Staubli VAL3: HM.pjx

--- HM.pjx ---
Parameters version=s7.8.2 stackSize=5000 millimeterUnit=true
Program file=JTPdemo.pgx
Program file=loadmaster0.pgx
Program file=loadmaster1.pgx
Program file=loadmaster2.pgx
Program file=loadmaster3.pgx
Program file=loadmaster4.pgx
Program file=loadmaster5.pgx
Program file=loadmaster6.pgx
Program file=loadmaster7.pgx
Program file=loadmaster8.pgx
Program file=loadmaster9.pgx
Program file=madol.pgx
Program file=oldmaduofrme.pgx
Program file=proDEMO.pgx
Program file=saveOldframe.pgx
Program file=SAVEtoolAfranme.pgx
Program file=SMOVE.pgx
Program file=start.pgx
Program file=stop.pgx
Program file=takestop.pgx
Program file=tooolAndFrame.pgx
Data file=HM.dtx
Library alias=master path=Disk://master/master.pjx
Library alias=lib path=Disk://frmtool/frmtool.pjx

--- HM.dtx ---
bool b0
bool b1 = true
bool b2
bool b3
bool b4
bool bA[10] = true
bool bPause
bool bruning
bool bstop
public dio diganying = {link=BasicIO-1\%I2}
dio distart = {link=usrIn0}
dio distop = {link=usrIn1}
dio ditab = {link=BasicIO-1\%I1}
dio dixi = {link=BasicIO-1\%I0}
dio dochui = {link=BasicIO-1\%Q0}
dio doxi = {link=BasicIO-1\%Q1}
public frame f1 = {x=112.060509, y=-257.129174, z=-98.62342, rx=-0.279882, ry=0.007961, rz=179.830294, fatherId=world[0]}
public frame frmaster[10]
  [0] = {x=487, y=64, z=-100.5, rx=5, rz=-92.998, fatherId=world[0]}
  [1] = {x=472, y=210, z=-97, rz=175, fatherId=world[0]}
  [2] = {x=472, y=201, z=-98, rx=0.5, rz=98, fatherId=world[0]}
  [3] = {fatherId=world[0]}
  [4] = {fatherId=world[0]}
  [5] = {fatherId=world[0]}
  [6] = {fatherId=world[0]}
  [7] = {x=487, y=64, z=-100.5, rx=5, rz=-92.998, fatherId=world[0]}
  [8] = {x=487, y=64, z=-100.5, rx=5, rz=-92.998, fatherId=world[0]}
  [9] = {x=487, y=64, z=-100.5, rx=5, rz=-92.998, fatherId=world[0]}
jointRx jA[20]
  [0] = {j1=-36.809158, j2=6.473103, j3=115.475326, j4=0.67904, j5=57.498227, j6=-129.910351}
  [1] = {j1=-46.642796, j2=10.279087, j3=109.084102, j4=6.799386, j5=57.689141, j6=-43.494821}
  [2] = {j1=-36.809158, j2=6.473103, j3=115.475326, j4=0.67904, j5=57.498227, j6=-129.910351}
  [3] = {j1=-46.642796, j2=10.279087, j3=109.084102, j4=6.799386, j5=57.689141, j6=-43.494821}
  [4] = {j1=-36.809158, j2=6.473103, j3=115.475326, j4=0.67904, j5=57.498227, j6=-129.910351}
  [5] = {j1=-46.642796, j2=10.279087, j3=109.084102, j4=6.799386, j5=57.689141, j6=-43.494821}
  [6] = {j1=-36.809158, j2=6.473103, j3=115.475326, j4=0.67904, j5=57.498227, j6=-129.910351}
  [7] = {j1=-46.642796, j2=10.279087, j3=109.084102, j4=6.799386, j5=57.689141, j6=-43.494821}
  [8] = {j1=-36.809158, j2=6.473103, j3=115.475326, j4=0.67904, j5=57.498227, j6=-129.910351}
  [9] = {j1=-46.642796, j2=10.279087, j3=109.084102, j4=6.799386, j5=57.689141, j6=-43.494821}
  [10] = {j1=-36.809158, j2=6.473103, j3=115.475326, j4=0.67904, j5=57.498227, j6=-129.910351}
  [11] = {j1=-46.642796, j2=10.279087, j3=109.084102, j4=6.799386, j5=57.689141, j6=-43.494821}
  [12] = {j1=-36.809158, j2=6.473103, j3=115.475326, j4=0.67904, j5=57.498227, j6=-129.910351}
  [13] = {j1=-46.642796, j2=10.279087, j3=109.084102, j4=6.799386, j5=57.689141, j6=-43.494821}
  [14] = {j1=-36.809158, j2=6.473103, j3=115.475326, j4=0.67904, j5=57.498227, j6=-129.910351}
  [15] = {j1=-46.642796, j2=10.279087, j3=109.084102, j4=6.799386, j5=57.689141, j6=-43.494821}
  [16] = {j1=-36.809158, j2=6.473103, j3=115.475326, j4=0.67904, j5=57.498227, j6=-129.910351}
  [17] = {j1=-46.642796, j2=10.279087, j3=109.084102, j4=6.799386, j5=57.689141, j6=-43.494821}
  [18] = {j1=-36.809158, j2=6.473103, j3=115.475326, j4=0.67904, j5=57.498227, j6=-129.910351}
  [19] = {j1=-46.642796, j2=10.279087, j3=109.084102, j4=6.799386, j5=57.689141, j6=-43.494821}
jointRx jXieLiao = {j1=-96.476357, j2=75.42768, j3=32.803482, j4=-0.025549, j5=71.586432, j6=-93.064419}
jointRx jbegin = {j1=-36.809158, j2=6.473103, j3=115.475326, j4=0.67904, j5=57.498227, j6=-129.910351}
jointRx jchack = {j1=-102.590963, j2=19.158438, j3=101.614955, j4=-0.038681, j5=59.106199, j6=77.212336}
jointRx jend = {j1=-46.642796, j2=10.279087, j3=109.084102, j4=6.799386, j5=57.689141, j6=-43.494821}
jointRx jf = {j1=-96.478721, j2=69.604961, j3=32.597072, j4=-0.024894, j5=77.614683, j6=-93.069451}
jointRx jready = {j1=-93.60071, j2=14.149819, j3=120.13944, j4=-0.061569, j5=45.526614, j6=86.705521}
jointRx jstart = {j1=-102.590964, j2=19.158205, j3=101.615123, j4=-0.038768, j5=59.105849, j6=77.212673}
mdesc m1
mdesc mFast
mdesc mSuDu[3]
  [0] = {leave=0.5, reach=0.5}
  [1] = {leave=0.5, reach=0.5}
  [2] = {leave=0.5, reach=0.5}
num n0 = 1
num n1 = 2
num n2
num nJTP
num nPY = 320
num nPYB
num nPYC = 320
num nPYtest = -0.957
num nPeak0[3]
  [0] = 66
  [1] = 198
num nPeak1[4]
  [0] = 193
  [1] = 359
  [2] = 551
num nPeak2
num nPeak3
num nPeak4
num nPeak5
num nPeak6
num nPeak7
num nPeak8
num nPeak9
num nc
num ndemo = 263
num nframe = 10
num nframeSave[10]
  [1] = 1
  [2] = 2
  [3] = 3
  [4] = 4
  [5] = 5
  [6] = 6
num ni
num ninttool = 10
num nmaster = 263
num nsize[10]
  [0] = 263
  [1] = 713
  [2] = 1183
num ntool = 10
num ntoolSave[10]
  [1] = 1
  [2] = 2
  [3] = 3
  [4] = 4
pointRx p1 = {x=0.01979, y=0.014228, z=76.837612, rx=0.284492, ry=-179.996615, rz=2.95459, fatherId=f1[0]}
pointRx p2 = {x=0.019785, y=0.014249, z=0.8, rx=0.28, ry=-179.997276, rz=2.954581, fatherId=f1[0]}
pointRx pXieLiao[2]
  [0] = {x=530.900904, y=-168.692362, z=119.392812, rx=179.999348, ry=-0.000559, rz=86.125781, fatherId=f1[0]}
  [1] = {x=530.900895, y=-168.692364, z=88.853022, rx=179.999359, ry=-0.000487, rz=86.125781, fatherId=f1[0]}
pointRx pdemo0[263]
  [0] = {x=-68.939309, y=2.594876, z=125.851419, rx=-179.999842, ry=-4.539241, rz=-20.572084, shoulder=lefty, elbow=epositive, wrist=wpositive, fatherId=frmaster[0]}
  [1] = {x=-70.093865, y=2.593252, z=111.351632, rx=179.999825, ry=-4.539343, rz=-20.573264, shoulder=lefty, elbow=epositive, wrist=wpositive, fatherId=frmaster[0]}
  [2] = {x=-70.092383, y=2.592813, z=101.346658, rx=179.998902, ry=-4.539362, rz=-20.572687, shoulder=lefty, elbow=epositive, wrist=wpositive, fatherId=frmaster[0]}
  [3] = {x=-65.564746, y=4.520144, z=104.636521, rx=-179.999623, ry=-7.320234, rz=-18.950696, shoulder=lefty, elbow=epositive, wrist=wpositive, fatherId=frmaster[0]}
  [4] = {x=-62.147679, y=5.718087, z=106.809457, rx=-179.999792, ry=-9.281495, rz=-17.978552, shoulder=lefty, elbow=epositive, wrist=wpositive, fatherId=frmaster[0]}
  [5] = {x=-57.8022, y=7.018139, z=109.291144, rx=179.999693, ry=-11.675298, rz=-16.93825, shoulder=lefty, elbow=epositive, wrist=wpositive, fatherId=frmaster[0]}
  [6] = {x=-55.21006, y=7.693586, z=110.648654, rx=-179.999664, ry=-13.066514, rz=-16.401657, shoulder=lefty, elbow=epositive, wrist=wpositive, fatherId=frmaster[0]}
  [7] = {x=-52.124031, y=8.434718, z=112.144392, rx=-179.999565, ry=-14.684361, rz=-15.820245, shoulder=lefty, elbow=epositive, wrist=wpositive, fatherId=frmaster[0]}
  [8] = {x=-48.559584, y=9.194588, z=113.730853, rx=179.999704, ry=-16.519257, rz=-15.226253, shoulder=lefty, elbow=epositive, wrist=wpositive, fatherId=frmaster[0]}
  [9] = {x=-44.443282, y=9.975646, z=115.393939, rx=-179.999788, ry=-18.600614, rz=-14.619836, shoulder=lefty, elbow=epositive, wrist=wpositive, fatherId=frmaster[0]}
  [10] = {x=-39.800946, y=10.739014, z=117.055469, rx=-179.999297, ry=-20.90861, rz=-14.028689, shoulder=lefty, elbow=epositive, wrist=wpositive, fatherId=frmaster[0]}
  [11] = {x=-34.573283, y=11.490434, z=118.675732, rx=-179.999727, ry=-23.468814, rz=-13.446694, shoulder=lefty, elbow=epositive, wrist=wpositive, fatherId=frmaster[0]}
  [12] = {x=-28.795169, y=12.206445, z=120.17003, rx=-179.99997, ry=-26.259293, rz=-12.893915, shoulder=lefty, elbow=epositive, wrist=wpositive, fatherId=frmaster[0]}
  [13] = {x=-25.703845, y=12.55415, z=120.847864, rx=-179.999289, ry=-27.738767, rz=-12.625116, shoulder=lefty, elbow=epositive, wrist=wpositive, fatherId=frmaster[0]}
  [14] = {x=-22.481958, y=12.893896, z=121.46453, rx=-179.999584, ry=-29.273016, rz=-12.362705, shoulder=lefty, elbow=epositive, wrist=wpositive, fatherId=frmaster[0]}
  [15] = {x=-19.100752, y=13.220332, z=122.011165, rx=179.999554, ry=-30.873819, rz=-12.110668, shoulder=lefty, elbow=epositive, wrist=wpositive, fatherId=frmaster[0]}
  [16] = {x=-15.56624, y=13.542118, z=122.492282, rx=179.999906, ry=-32.542669, rz=-11.862432, shoulder=lefty, elbow=epositive, wrist=wpositive, fatherId=frmaster[0]}
  [17] = {x=-11.862171, y=13.86112, z=122.876566, rx=-179.999624, ry=-34.280739, rz=-11.617025, shoulder=lefty, elbow=epositive, wrist=wpositive, fatherId=frmaster[0]}
  [18] = {x=-7.999903, y=14.172788, z=123.156947, rx=-179.999236, ry=-36.08968, rz=-11.375401, shoulder=lefty, elbow=epositive, wrist=wpositive, fatherId=frmaster[0]}
  [19] = {x=-3.982068, y=14.472199, z=123.31508, rx=-179.999527, ry=-37.973145, rz=-11.146259, shoulder=lefty, elbow=epositive, wrist=wpositive, fatherId=frmaster[0]}
  [20] = {x=0.003718, y=14.757289, z=123.343316, rx=-179.999752, ry=-39.835809, rz=-10.926527, shoulder=lefty, elbow=epositive, wrist=wpositive, fatherId=frmaster[0]}
  [21] = {x=3.926135, y=15.026312, z=123.249243, rx=-179.999627, ry=-41.673849, rz=-10.71735, shoulder=lefty, elbow=epositive, wrist=wpositive, fatherId=frmaster[0]}
  [22] = {x=7.787882, y=15.285683, z=123.023611, rx=-179.999358, ry=-43.485441, rz=-10.516961, shoulder=lefty, elbow=epositive, wrist=wpositive, fatherId=frmaster[0]}
  [23] = {x=3.636586, y=13.055492, z=123.517209, rx=-179.999236, ry=-41.68691, rz=-12.371075, shoulder=lefty, elbow=epositive, wrist=wpositive, fatherId=frmaster[0]}
  [24] = {x=-0.115648, y=10.554981, z=123.842224, rx=-179.9989, ry=-40.072666, rz=-14.410733, shoulder=lefty, elbow=epositive, wrist=wpositive, fatherId=frmaster[0]}
  [25] = {x=-2.87591, y=7.781393, z=124.033861, rx=-179.999939, ry=-38.90966, rz=-16.64011, shoulder=lefty, elbow=epositive, wrist=wpositive, fatherId=frmaster[0]}
  [26] = {x=-5.00539, y=4.722334, z=124.137637, rx=-179.999391, ry=-38.009486, rz=-19.063272, shoulder=lefty, elbow=epositive, wrist=wpositive, fatherId=frmaster[0]}
  [27] = {x=-6.286632, y=1.407733, z=124.172868, rx=-179.999461, ry=-37.465687, rz=-21.663049, shoulder=lefty, elbow=epositive, wrist=wpositive, fatherId=frmaster[0]}
  [28] = {x=-6.757242, y=-1.994395, z=124.137734, rx=-179.999849, ry=-37.245975, rz=-24.324062, shoulder=lefty, elbow=epositive, wrist=wpositive, fatherId=frmaster[0]}
  [29] = {x=-6.623, y=-5.406644, z=124.030721, rx=-179.999523, ry=-37.25052, rz=-26.994443, shoulder=lefty, elbow=epositive, wrist=wpositive, fatherId=frmaster[0]}
  [30] = {x=-5.670017, y=-8.784356, z=123.866129, rx=179.999811, ry=-37.580919, rz=-29.6487, shoulder=lefty, elbow=epositive, wrist=wpositive, fatherId=frmaster[0]}
  [31] = {x=-4.463415, y=-12.188788, z=123.606311, rx=-179.999254, ry=-37.973613, rz=-32.334872, shoulder=lefty, elbow=epositive, wrist=wpositive, fatherId=frmaster[0]}
  [32] = {x=-2.488328, y=-15.635885, z=123.233005, rx=-179.999282, ry=-38.667419, rz=-35.069863, shoulder=lefty, elbow=epositive, wrist=wpositive, fatherId=frmaster[0]}
  [33] = {x=-0.694211, y=-19.173546, z=122.713263, rx=-179.99927, ry=-39.206278, rz=-37.895277, shoulder=lefty, elbow=epositive, wrist=wpositive, fatherId=frmaster[0]}
  [34] = {x=1.757246, y=-22.68427, z=122.039686, rx=179.999513, ry=-40.003209, rz=-40.732797, shoulder=lefty, elbow=epositive, wrist=wpositive, fatherId=frmaster[0]}
  [35] = {x=3.612463, y=-26.090704, z=121.2463, rx=-179.999323, ry=-40.461466, rz=-43.533179, shoulder=lefty, elbow=epositive, wrist=wpositive, fatherId=frmaster[0]}
  [36] = {x=6.005382, y=-29.344396, z=120.330355, rx=-179.999297, ry=-41.144506, rz=-46.26609, shoulder=lefty, elbow=epositive, wrist=wpositive, fatherId=frmaster[0]}
  [37] = {x=8.178744, y=-32.51397, z=119.292757, rx=-179.999423, ry=-41.674458, rz=-48.980771, shoulder=lefty, elbow=epositive, wrist=wpositive, fatherId=frmaster[0]}
  [38] = {x=10.802026, y=-35.564113, z=118.108689, rx=-179.999959, ry=-42.396715, rz=-51.657334, shoulder=lefty, elbow=epositive, wrist=wpositive, fatherId=frmaster[0]}
  [39] = {x=13.535281, y=-38.529801, z=116.777056, rx=179.9997, ry=-43.139921, rz=-54.32829, shoulder=lefty, elbow=epositive, wrist=wpositive, fatherId=frmaster[0]}
  [40] = {x=16.594916, y=-41.383811, z=115.276942, rx=-179.999131, ry=-44.02302, rz=-56.968323, shoulder=lefty, elbow=epositive, wrist=wpositive, fatherId=frmaster[0]}
  [41] = {x=19.918159, y=-44.039781, z=113.620021, rx=-179.999247, ry=-45.050326, rz=-59.514928, shoulder=lefty, elbow=epositive, wrist=wpositive, fatherId=frmaster[0]}
  [42] = {x=23.337445, y=-46.461139, z=111.840864, rx=179.999666, ry=-46.157544, rz=-61.921405, shoulder=lefty, elbow=epositive, wrist=wpositive, fatherId=frmaster[0]}
  [43] = {x=19.98531, y=-46.203057, z=112.638501, rx=-179.999542, ry=-44.473252, rz=-61.637393, shoulder=lefty, elbow=epositive, wrist=wpositive, fatherId=frmaster[0]}
  [44] = {x=16.475747, y=-45.923809, z=113.355993, rx=-179.999849, ry=-42.732145, rz=-61.337507, shoulder=lefty, elbow=epositive, wrist=wpositive, fatherId=frmaster[0]}
  [45] = {x=12.814869, y=-45.622369, z=113.989509, rx=179.999801, ry=-40.928708, rz=-61.018055, shoulder=lefty, elbow=epositive, wrist=wpositive, fatherId=frmaster[0]}
  [46] = {x=8.994815, y=-45.291604, z=114.523598, rx=-179.998902, ry=-39.065668, rz=-60.674105, shoulder=lefty, elbow=epositive, wrist=wpositive, fatherId=frmaster[0]}
  [47] = {x=5.221971, y=-44.883621, z=114.948885, rx=179.99941, ry=-37.262806, rz=-60.255183, shoulder=lefty, elbow=epositive, wrist=wpositive, fatherId=frmaster[0]}
  [48] = {x=1.449749, y=-44.426571, z=115.268039, rx=-179.999677, ry=-35.476818, rz=-59.799009, shoulder=lefty, elbow=epositive, wrist=wpositive, fatherId=frmaster[0]}
  [49] = {x=-2.30993, y=-43.925823, z=115.469722, rx=-179.999667, ry=-33.714009, rz=-59.302848, shoulder=lefty, elbow=epositive, wrist=wpositive, fatherId=frmaster[0]}
  [50] = {x=-6.054682, y=-43.371912, z=115.566057, rx=-179.99921, ry=-31.979643, rz=-58.765546, shoulder=lefty, elbow=epositive, wrist=wpositive, fatherId=frmaster[0]}
  [51] = {x=-9.706723, y=-42.74106, z=115.566586, rx=-179.999762, ry=-30.311063, rz=-58.161529, shoulder=lefty, elbow=epositive, wrist=wpositive, fatherId=frmaster[0]}
  [52] = {x=-13.324451, y=-42.074603, z=115.473731, rx=179.999869, ry=-28.675999, rz=-57.526544, shoulder=lefty, elbow=epositive, wrist=wpositive, fatherId=frmaster[0]}
  [53] = {x=-16.85983, y=-41.366634, z=115.277163, rx=179.999422, ry=-27.08369, rz=-56.861863, shoulder=lefty, elbow=epositive, wrist=wpositive, fatherId=frmaster[0]}
  [54] = {x=-20.301815, y=-40.617438, z=115.002996, rx=-179.999332, ry=-25.546739, rz=-56.16562, shoulder=lefty, elbow=epositive, wrist=wpositive, fatherId=frmaster[0]}
  [55] = {x=-26.791225, y=-38.992184, z=114.248958, rx=-179.998983, ry=-22.681622, rz=-54.674543, shoulder=lefty, elbow=epositive, wrist=wpositive, fatherId=frmaster[0]}
  [56] = {x=-32.776952, y=-37.211639, z=113.279864, rx=179.999314, ry=-20.079214, rz=-53.068219, shoulder=lefty, elbow=epositive, wrist=wpositive, fatherId=frmaster[0]}
  [57] = {x=-38.202715, y=-35.254548, z=112.201778, rx=-179.999362, ry=-17.75731, rz=-51.337224, shoulder=lefty, elbow=epositive, wrist=wpositive, fatherId=frmaster[0]}
  [58] = {x=-43.075297, y=-33.139465, z=111.069332, rx=-179.99912, ry=-15.713738, rz=-49.495669, shoulder=lefty, elbow=epositive, wrist=wpositive, fatherId=frmaster[0]}
  [59] = {x=-47.485041, y=-30.827965, z=109.907709, rx=-179.999984, ry=-13.891332, rz=-47.517107, shoulder=lefty, elbow=epositive, wrist=wpositive, fatherId=frmaster[0]}
  [60] = {x=-51.464947, y=-28.297069, z=108.771217, rx=-179.999297, ry=-12.28541, rz=-45.387575, shoulder=lefty, elbow=epositive, wrist=wpositive, fatherId=frmaster[0]}
  [61] = {x=-58.258069, y=-22.435578, z=106.618321, rx=179.999827, ry=-9.619917, rz=-40.577437, shoulder=lefty, elbow=epositive, wrist=wpositive, fatherId=frmaster[0]}
  [62] = {x=-63.471689, y=-15.637158, z=104.757087, rx=179.999576, ry=-7.611857, rz=-35.15207, shoulder=lefty, elbow=epositive, wrist=wpositive, fatherId=frmaster[0]}
  [63] = {x=-69.230412, y=-4.124169, z=101.957036, rx=-179.999606, ry=-5.040121, rz=-25.997789, shoulder=lefty, elbow=epositive, wrist=wpositive, fatherId=frmaster[0]}
  [64] = {x=-69.233338, y=-4.126295, z=111.947543, rx=179.999548, ry=-5.039948, rz=-25.997986, shoulder=lefty, elbow=epositive, wrist=wpositive, fatherId=frmaster[0]}
  [65] = {x=-67.950588, y=-4.124727, z=126.453883, rx=179.999566, ry=-5.039306, rz=-25.997643, shoulder=lefty, elbow=epositive, wrist=wpositive, fatherId=frmaster[0]}
  [66] = {x=-68.939309, y=2.594876, z=125.851419, rx=0.000158, ry=-175.460759, rz=-20.572084, shoulder=lefty, elbow=epositive, wrist=wpositive, fatherId=frmaster[0]}
  [67] = {x=-70.093865, y=2.593252, z=111.351632, rx=-0.000175, ry=-175.460657, rz=-20.573264, shoulder=lefty, elbow=epositive, wrist=wpositive, fatherId=frmaster[0]}
  [68] = {x=-70.092383, y=2.592813, z=101.346658, rx=-0.001098, ry=-175.460638, rz=-20.572687, shoulder=lefty, elbow=epositive, wrist=wpositive, fatherId=frmaster[0]}
  [69] = {x=-65.564746, y=4.520144, z=104.636521, rx=0.000377, ry=-172.679766, rz=-18.950696, shoulder=lefty, elbow=epositive, wrist=wpositive, fatherId=frmaster[0]}
  [70] = {x=-62.147679, y=5.718087, z=106.809457, rx=0.000208, ry=-170.718505, rz=-17.978552, shoulder=lefty, elbow=epositive, wrist=wpositive, fatherId=frmaster[0]}
  [71] = {x=-57.8022, y=7.018139, z=109.291144, rx=-0.000307, ry=-168.324702, rz=-16.93825, shoulder=lefty, elbow=epositive, wrist=wpositive, fatherId=frmaster[0]}
  [72] = {x=-55.21006, y=7.693586, z=110.648654, rx=0.000336, ry=-166.933486, rz=-16.401657, shoulder=lefty, elbow=epositive, wrist=wpositive, fatherId=frmaster[0]}
  [73] = {x=-52.124031, y=8.434718, z=112.144392, rx=0.000435, ry=-165.315639, rz=-15.820245, shoulder=lefty, elbow=epositive, wrist=wpositive, fatherId=frmaster[0]}
  [74] = {x=-48.559584, y=9.194588, z=113.730853, rx=-0.000296, ry=-163.480743, rz=-15.226253, shoulder=lefty, elbow=epositive, wrist=wpositive, fatherId=frmaster[0]}
  [75] = {x=-44.443282, y=9.975646, z=115.393939, rx=0.000212, ry=-161.399386, rz=-14.619836, shoulder=lefty, elbow=epositive, wrist=wpositive, fatherId=frmaster[0]}
  [76] = {x=-39.800946, y=10.739014, z=117.055469, rx=0.000703, ry=-159.09139, rz=-14.028689, shoulder=lefty, elbow=epositive, wrist=wpositive, fatherId=frmaster[0]}
  [77] = {x=-34.573283, y=11.490434, z=118.675732, rx=0.000273, ry=-156.531186, rz=-13.446694, shoulder=lefty, elbow=epositive, wrist=wpositive, fatherId=frmaster[0]}
  [78] = {x=-28.795169, y=12.206445, z=120.17003, rx=0.00003, ry=-153.740707, rz=-12.893915, shoulder=lefty, elbow=epositive, wrist=wpositive, fatherId=frmaster[0]}
  [79] = {x=-25.703845, y=12.55415, z=120.847864, rx=0.000711, ry=-152.261233, rz=-12.625116, shoulder=lefty, elbow=epositive, wrist=wpositive, fatherId=frmaster[0]}
  [80] = {x=-22.481958, y=12.893896, z=121.46453, rx=0.000416, ry=-150.726984, rz=-12.362705, shoulder=lefty, elbow=epositive, wrist=wpositive, fatherId=frmaster[0]}
  [81] = {x=-19.100752, y=13.220332, z=122.011165, rx=-0.000446, ry=-149.126181, rz=-12.110668, shoulder=lefty, elbow=epositive, wrist=wpositive, fatherId=frmaster[0]}
  [82] = {x=-15.56624, y=13.542118, z=122.492282, rx=-0.000094, ry=-147.457331, rz=-11.862432, shoulder=lefty, elbow=epositive, wrist=wpositive, fatherId=frmaster[0]}
  [83] = {x=-11.862171, y=13.86112, z=122.876566, rx=0.000376, ry=-145.719261, rz=-11.617025, shoulder=lefty, elbow=epositive, wrist=wpositive, fatherId=frmaster[0]}
  [84] = {x=-7.999903, y=14.172788, z=123.156947, rx=0.000764, ry=-143.91032, rz=-11.375401, shoulder=lefty, elbow=epositive, wrist=wpositive, fatherId=frmaster[0]}
  [85] = {x=-3.982068, y=14.472199, z=123.31508, rx=0.000473, ry=-142.026855, rz=-11.146259, shoulder=lefty, elbow=epositive, wrist=wpositive, fatherId=frmaster[0]}
  [86] = {x=0.003718, y=14.757289, z=123.343316, rx=0.000248, ry=-140.164191, rz=-10.926527, shoulder=lefty, elbow=epositive, wrist=wpositive, fatherId=frmaster[0]}
  [87] = {x=3.926135, y=15.026312, z=123.249243, rx=0.000373, ry=-138.326151, rz=-10.71735, shoulder=lefty, elbow=epositive, wrist=wpositive, fatherId=frmaster[0]}
  [88] = {x=7.787882, y=15.285683, z=123.023611, rx=0.000642, ry=-136.514559, rz=-10.516961, shoulder=lefty, elbow=epositive, wrist=wpositive, fatherId=frmaster[0]}
  [89] = {x=3.636586, y=13.055492, z=123.517209, rx=0.000764, ry=-138.31309, rz=-12.371075, shoulder=lefty, elbow=epositive, wrist=wpositive, fatherId=frmaster[0]}
  [90] = {x=-0.115648, y=10.554981, z=123.842224, rx=0.0011, ry=-139.927334, rz=-14.410733, shoulder=lefty, elbow=epositive, wrist=wpositive, fatherId=frmaster[0]}
  [91] = {x=-2.87591, y=7.781393, z=124.033861, rx=0.000061, ry=-141.09034, rz=-16.64011, shoulder=lefty, elbow=epositive, wrist=wpositive, fatherId=frmaster[0]}
  [92] = {x=-5.00539, y=4.722334, z=124.137637, rx=0.000609, ry=-141.990514, rz=-19.063272, shoulder=lefty, elbow=epositive, wrist=wpositive, fatherId=frmaster[0]}
  [93] = {x=-6.286632, y=1.407733, z=124.172868, rx=0.000539, ry=-142.534313, rz=-21.663049, shoulder=lefty, elbow=epositive, wrist=wpositive, fatherId=frmaster[0]}
  [94] = {x=-6.757242, y=-1.994395, z=124.137734, rx=0.000151, ry=-142.754025, rz=-24.324062, shoulder=lefty, elbow=epositive, wrist=wpositive, fatherId=frmaster[0]}
  [95] = {x=-6.623, y=-5.406644, z=124.030721, rx=0.000477, ry=-142.74948, rz=-26.994443, shoulder=lefty, elbow=epositive, wrist=wpositive, fatherId=frmaster[0]}
  [96] = {x=-5.670017, y=-8.784356, z=123.866129, rx=-0.000189, ry=-142.419081, rz=-29.6487, shoulder=lefty, elbow=epositive, wrist=wpositive, fatherId=frmaster[0]}
  [97] = {x=-4.463415, y=-12.188788, z=123.606311, rx=0.000746, ry=-142.026387, rz=-32.334872, shoulder=lefty, elbow=epositive, wrist=wpositive, fatherId=frmaster[0]}
  [98] = {x=-2.488328, y=-15.635885, z=123.233005, rx=0.000718, ry=-141.332581, rz=-35.069863, shoulder=lefty, elbow=epositive, wrist=wpositive, fatherId=frmaster[0]}
  [99] = {x=-0.694211, y=-19.173546, z=122.713263, rx=0.00073, ry=-140.793722, rz=-37.895277, shoulder=lefty, elbow=epositive, wrist=wpositive, fatherId=frmaster[0]}
  [100] = {x=1.757246, y=-22.68427, z=122.039686, rx=-0.000487, ry=-139.996791, rz=-40.732797, shoulder=lefty, elbow=epositive, wrist=wpositive, fatherId=frmaster[0]}
  [101] = {x=3.612463, y=-26.090704, z=121.2463, rx=0.000677, ry=-139.538534, rz=-43.533179, shoulder=lefty, elbow=epositive, wrist=wpositive, fatherId=frmaster[0]}
  [102] = {x=6.005382, y=-29.344396, z=120.330355, rx=0.000703, ry=-138.855494, rz=-46.26609, shoulder=lefty, elbow=epositive, wrist=wpositive, fatherId=frmaster[0]}
  [103] = {x=8.178744, y=-32.51397, z=119.292757, rx=0.000577, ry=-138.325542, rz=-48.980771, shoulder=lefty, elbow=epositive, wrist=wpositive, fatherId=frmaster[0]}
  [104] = {x=10.802026, y=-35.564113, z=118.108689, rx=0.000041, ry=-137.603285, rz=-51.657334, shoulder=lefty, elbow=epositive, wrist=wpositive, fatherId=frmaster[0]}
  [105] = {x=13.535281, y=-38.529801, z=116.777056, rx=-0.0003, ry=-136.860079, rz=-54.32829, shoulder=lefty, elbow=epositive, wrist=wpositive, fatherId=frmaster[0]}
  [106] = {x=16.594916, y=-41.383811, z=115.276942, rx=0.000869, ry=-135.97698, rz=-56.968323, shoulder=lefty, elbow=epositive, wrist=wpositive, fatherId=frmaster[0]}
  [107] = {x=19.918159, y=-44.039781, z=113.620021, rx=0.000753, ry=-134.949674, rz=-59.514928, shoulder=lefty, elbow=epositive, wrist=wpositive, fatherId=frmaster[0]}
  [108] = {x=23.337445, y=-46.461139, z=111.840864, rx=-0.000334, ry=-133.842456, rz=-61.921405, shoulder=lefty, elbow=epositive, wrist=wpositive, fatherId=frmaster[0]}
  [109] = {x=19.98531, y=-46.203057, z=112.638501, rx=0.000458, ry=-135.526748, rz=-61.637393, shoulder=lefty, elbow=epositive, wrist=wpositive, fatherId=frmaster[0]}
  [110] = {x=16.475747, y=-45.923809, z=113.355993, rx=0.000151, ry=-137.267855, rz=-61.337507, shoulder=lefty, elbow=epositive, wrist=wpositive, fatherId=frmaster[0]}
  [111] = {x=12.814869, y=-45.622369, z=113.989509, rx=-0.000199, ry=-139.071292, rz=-61.018055, shoulder=lefty, elbow=epositive, wrist=wpositive, fatherId=frmaster[0]}
  [112] = {x=8.994815, y=-45.291604, z=114.523598, rx=0.001098, ry=-140.934332, rz=-60.674105, shoulder=lefty, elbow=epositive, wrist=wpositive, fatherId=frmaster[0]}
  [113] = {x=5.221971, y=-44.883621, z=114.948885, rx=-0.00059, ry=-142.737194, rz=-60.255183, shoulder=lefty, elbow=epositive, wrist=wpositive, fatherId=frmaster[0]}
  [114] = {x=1.449749, y=-44.426571, z=115.268039, rx=0.000323, ry=-144.523182, rz=-59.799009, shoulder=lefty, elbow=epositive, wrist=wpositive, fatherId=frmaster[0]}
  [115] = {x=-2.30993, y=-43.925823, z=115.469722, rx=0.000333, ry=-146.285991, rz=-59.302848, shoulder=lefty, elbow=epositive, wrist=wpositive, fatherId=frmaster[0]}
  [116] = {x=-6.054682, y=-43.371912, z=115.566057, rx=0.00079, ry=-148.020357, rz=-58.765546, shoulder=lefty, elbow=epositive, wrist=wpositive, fatherId=frmaster[0]}
  [117] = {x=-9.706723, y=-42.74106, z=115.566586, rx=0.000238, ry=-149.688937, rz=-58.161529, shoulder=lefty, elbow=epositive, wrist=wpositive, fatherId=frmaster[0]}
  [118] = {x=-13.324451, y=-42.074603, z=115.473731, rx=-0.000131, ry=-151.324001, rz=-57.526544, shoulder=lefty, elbow=epositive, wrist=wpositive, fatherId=frmaster[0]}
  [119] = {x=-16.85983, y=-41.366634, z=115.277163, rx=-0.000578, ry=-152.91631, rz=-56.861863, shoulder=lefty, elbow=epositive, wrist=wpositive, fatherId=frmaster[0]}
  [120] = {x=-20.301815, y=-40.617438, z=115.002996, rx=0.000668, ry=-154.453261, rz=-56.16562, shoulder=lefty, elbow=epositive, wrist=wpositive, fatherId=frmaster[0]}
  [121] = {x=-26.791225, y=-38.992184, z=114.248958, rx=0.001017, ry=-157.318378, rz=-54.674543, shoulder=lefty, elbow=epositive, wrist=wpositive, fatherId=frmaster[0]}
  [122] = {x=-32.776952, y=-37.211639, z=113.279864, rx=-0.000686, ry=-159.920786, rz=-53.068219, shoulder=lefty, elbow=epositive, wrist=wpositive, fatherId=frmaster[0]}
  [123] = {x=-38.202715, y=-35.254548, z=112.201778, rx=0.000638, ry=-162.24269, rz=-51.337224, shoulder=lefty, elbow=epositive, wrist=wpositive, fatherId=frmaster[0]}
  [124] = {x=-43.075297, y=-33.139465, z=111.069332, rx=0.00088, ry=-164.286262, rz=-49.495669, shoulder=lefty, elbow=epositive, wrist=wpositive, fatherId=frmaster[0]}
  [125] = {x=-47.485041, y=-30.827965, z=109.907709, rx=0.000016, ry=-166.108668, rz=-47.517107, shoulder=lefty, elbow=epositive, wrist=wpositive, fatherId=frmaster[0]}
  [126] = {x=-51.464947, y=-28.297069, z=108.771217, rx=0.000703, ry=-167.71459, rz=-45.387575, shoulder=lefty, elbow=epositive, wrist=wpositive, fatherId=frmaster[0]}
  [127] = {x=-58.258069, y=-22.435578, z=106.618321, rx=-0.000173, ry=-170.380083, rz=-40.577437, shoulder=lefty, elbow=epositive, wrist=wpositive, fatherId=frmaster[0]}
  [128] = {x=-63.471689, y=-15.637158, z=104.757087, rx=-0.000424, ry=-172.388143, rz=-35.15207, shoulder=lefty, elbow=epositive, wrist=wpositive, fatherId=frmaster[0]}
  [129] = {x=-69.230412, y=-4.124169, z=101.957036, rx=0.000394, ry=-174.959879, rz=-25.997789, shoulder=lefty, elbow=epositive, wrist=wpositive, fatherId=frmaster[0]}
  [130] = {x=-69.233338, y=-4.126295, z=111.947543, rx=-0.000452, ry=-174.960052, rz=-25.997986, shoulder=lefty, elbow=epositive, wrist=wpositive, fatherId=frmaster[0]}
  [131] = {x=-67.950588, y=-4.124727, z=126.453883, rx=-0.000434, ry=-174.960694, rz=-25.997643, shoulder=lefty, elbow=epositive, wrist=wpositive, fatherId=frmaster[0]}
  [132] = {x=-68.941187, y=-2.594666, z=125.851852, rx=0.000032, ry=-175.461039, rz=20.573522, shoulder=lefty, elbow=epositive, wrist=wpositive, fatherId=frmaster[0]}
  [133] = {x=-70.091269, y=-2.592516, z=111.352514, rx=0.000846, ry=-175.461111, rz=20.573541, shoulder=lefty, elbow=epositive, wrist=wpositive, fatherId=frmaster[0]}
  [134] = {x=-70.091245, y=-2.592615, z=101.352, rx=0.000033, ry=-175.460833, rz=20.573205, shoulder=lefty, elbow=epositive, wrist=wpositive, fatherId=frmaster[0]}
  [135] = {x=-65.560701, y=-4.52076, z=104.634327, rx=-0.000281, ry=-172.679563, rz=18.95207, shoulder=lefty, elbow=epositive, wrist=wpositive, fatherId=frmaster[0]}
  [136] = {x=-62.144277, y=-5.717504, z=106.803129, rx=-0.000359, ry=-170.718649, rz=17.978978, shoulder=lefty, elbow=epositive, wrist=wpositive, fatherId=frmaster[0]}
  [137] = {x=-57.806655, y=-7.017721, z=109.289468, rx=-0.000663, ry=-168.324759, rz=16.938409, shoulder=lefty, elbow=epositive, wrist=wpositive, fatherId=frmaster[0]}
  [138] = {x=-55.21076, y=-7.694538, z=110.650126, rx=-0.000407, ry=-166.933915, rz=16.401878, shoulder=lefty, elbow=epositive, wrist=wpositive, fatherId=frmaster[0]}
  [139] = {x=-52.128732, y=-8.432815, z=112.151089, rx=0.000619, ry=-165.315499, rz=15.82104, shoulder=lefty, elbow=epositive, wrist=wpositive, fatherId=frmaster[0]}
  [140] = {x=-48.562509, y=-9.195661, z=113.731399, rx=-0.000489, ry=-163.480823, rz=15.226365, shoulder=lefty, elbow=epositive, wrist=wpositive, fatherId=frmaster[0]}
  [141] = {x=-44.445238, y=-9.974206, z=115.393252, rx=0.000319, ry=-161.400136, rz=14.620936, shoulder=lefty, elbow=epositive, wrist=wpositive, fatherId=frmaster[0]}
  [142] = {x=-39.805042, y=-10.739339, z=117.051018, rx=-0.000573, ry=-159.090853, rz=14.030338, shoulder=lefty, elbow=epositive, wrist=wpositive, fatherId=frmaster[0]}
  [143] = {x=-34.571504, y=-11.488063, z=118.672785, rx=0.000897, ry=-156.530797, rz=13.448615, shoulder=lefty, elbow=epositive, wrist=wpositive, fatherId=frmaster[0]}
  [144] = {x=-28.796804, y=-12.205792, z=120.171192, rx=0.000075, ry=-153.741262, rz=12.893974, shoulder=lefty, elbow=epositive, wrist=wpositive, fatherId=frmaster[0]}
  [145] = {x=-25.705389, y=-12.553736, z=120.842951, rx=0.000084, ry=-152.260896, rz=12.626325, shoulder=lefty, elbow=epositive, wrist=wpositive, fatherId=frmaster[0]}
  [146] = {x=-22.482081, y=-12.893063, z=121.465163, rx=0.000714, ry=-150.7265, rz=12.362432, shoulder=lefty, elbow=epositive, wrist=wpositive, fatherId=frmaster[0]}
  [147] = {x=-19.099649, y=-13.220159, z=122.01174, rx=0.000074, ry=-149.12637, rz=12.11146, shoulder=lefty, elbow=epositive, wrist=wpositive, fatherId=frmaster[0]}
  [148] = {x=-15.563891, y=-13.544095, z=122.485202, rx=-0.000697, ry=-147.457564, rz=11.862282, shoulder=lefty, elbow=epositive, wrist=wpositive, fatherId=frmaster[0]}
  [149] = {x=-11.860292, y=-13.859789, z=122.869811, rx=-0.000343, ry=-145.71961, rz=11.617688, shoulder=lefty, elbow=epositive, wrist=wpositive, fatherId=frmaster[0]}
  [150] = {x=-7.999201, y=-14.170821, z=123.152049, rx=0.0007, ry=-143.910847, rz=11.376413, shoulder=lefty, elbow=epositive, wrist=wpositive, fatherId=frmaster[0]}
  [151] = {x=-3.976731, y=-14.469679, z=123.320363, rx=0.001797, ry=-142.026592, rz=11.147405, shoulder=lefty, elbow=epositive, wrist=wpositive, fatherId=frmaster[0]}
  [152] = {x=-0.001611, y=-14.755184, z=123.349313, rx=0.000787, ry=-140.164211, rz=10.926322, shoulder=lefty, elbow=epositive, wrist=wpositive, fatherId=frmaster[0]}
  [153] = {x=3.921658, y=-15.027909, z=123.245131, rx=-0.000507, ry=-138.325584, rz=10.717247, shoulder=lefty, elbow=epositive, wrist=wpositive, fatherId=frmaster[0]}
  [154] = {x=7.787656, y=-15.282792, z=123.030151, rx=0.001801, ry=-136.514, rz=10.518616, shoulder=lefty, elbow=epositive, wrist=wpositive, fatherId=frmaster[0]}
  [155] = {x=3.632632, y=-13.0539, z=123.518074, rx=-0.00005, ry=-138.313563, rz=12.370731, shoulder=lefty, elbow=epositive, wrist=wpositive, fatherId=frmaster[0]}
  [156] = {x=-0.116628, y=-10.553936, z=123.837966, rx=0.000032, ry=-139.927576, rz=14.411441, shoulder=lefty, elbow=epositive, wrist=wpositive, fatherId=frmaster[0]}
  [157] = {x=-2.870576, y=-7.779605, z=124.040599, rx=0.000895, ry=-141.090255, rz=16.640287, shoulder=lefty, elbow=epositive, wrist=wpositive, fatherId=frmaster[0]}
  [158] = {x=-5.004213, y=-4.719529, z=124.142877, rx=0.001306, ry=-141.990068, rz=19.065288, shoulder=lefty, elbow=epositive, wrist=wpositive, fatherId=frmaster[0]}
  [159] = {x=-6.286234, y=-1.405857, z=124.170085, rx=0.000925, ry=-142.534454, rz=21.665507, shoulder=lefty, elbow=epositive, wrist=wpositive, fatherId=frmaster[0]}
  [160] = {x=-6.763491, y=1.995044, z=124.139406, rx=0.000204, ry=-142.753566, rz=24.324557, shoulder=lefty, elbow=epositive, wrist=wpositive, fatherId=frmaster[0]}
  [161] = {x=-6.628353, y=5.404754, z=124.035693, rx=-0.000517, ry=-142.749254, rz=26.994765, shoulder=lefty, elbow=epositive, wrist=wpositive, fatherId=frmaster[0]}
  [162] = {x=-5.669968, y=8.784748, z=123.870598, rx=0.000973, ry=-142.419688, rz=29.65073, shoulder=lefty, elbow=epositive, wrist=wpositive, fatherId=frmaster[0]}
  [163] = {x=-4.462138, y=12.188846, z=123.600895, rx=-0.000123, ry=-142.026144, rz=32.334503, shoulder=lefty, elbow=epositive, wrist=wpositive, fatherId=frmaster[0]}
  [164] = {x=-2.489646, y=15.635578, z=123.227559, rx=-0.001174, ry=-141.332529, rz=35.069591, shoulder=lefty, elbow=epositive, wrist=wpositive, fatherId=frmaster[0]}
  [165] = {x=-0.697365, y=19.173794, z=122.703604, rx=-0.000361, ry=-140.794344, rz=37.895465, shoulder=lefty, elbow=epositive, wrist=wpositive, fatherId=frmaster[0]}
  [166] = {x=1.761902, y=22.681657, z=122.038748, rx=0.000171, ry=-139.996822, rz=40.733105, shoulder=lefty, elbow=epositive, wrist=wpositive, fatherId=frmaster[0]}
  [167] = {x=3.610937, y=26.090403, z=121.250151, rx=0.000058, ry=-139.538873, rz=43.535028, shoulder=lefty, elbow=epositive, wrist=wpositive, fatherId=frmaster[0]}
  [168] = {x=6.005086, y=29.344743, z=120.329381, rx=0.000524, ry=-138.855396, rz=46.265313, shoulder=lefty, elbow=epositive, wrist=wpositive, fatherId=frmaster[0]}
  [169] = {x=8.175238, y=32.513013, z=119.28988, rx=-0.000185, ry=-138.325721, rz=48.981987, shoulder=lefty, elbow=epositive, wrist=wpositive, fatherId=frmaster[0]}
  [170] = {x=10.804669, y=35.563809, z=118.108795, rx=0.000305, ry=-137.603007, rz=51.657982, shoulder=lefty, elbow=epositive, wrist=wpositive, fatherId=frmaster[0]}
  [171] = {x=13.537862, y=38.530039, z=116.77667, rx=-0.000277, ry=-136.85975, rz=54.327489, shoulder=lefty, elbow=epositive, wrist=wpositive, fatherId=frmaster[0]}
  [172] = {x=16.594305, y=41.382503, z=115.269063, rx=0.000224, ry=-135.977587, rz=56.970299, shoulder=lefty, elbow=epositive, wrist=wpositive, fatherId=frmaster[0]}
  [173] = {x=19.918306, y=44.041072, z=113.61946, rx=0.000951, ry=-134.949818, rz=59.514719, shoulder=lefty, elbow=epositive, wrist=wpositive, fatherId=frmaster[0]}
  [174] = {x=23.334897, y=46.459403, z=111.834207, rx=-0.001026, ry=-133.842409, rz=61.920851, shoulder=lefty, elbow=epositive, wrist=wpositive, fatherId=frmaster[0]}
  [175] = {x=19.980834, y=46.20086, z=112.638726, rx=-0.000058, ry=-135.526892, rz=61.638901, shoulder=lefty, elbow=epositive, wrist=wpositive, fatherId=frmaster[0]}
  [176] = {x=16.481484, y=45.924464, z=113.358772, rx=0.000845, ry=-137.268507, rz=61.33928, shoulder=lefty, elbow=epositive, wrist=wpositive, fatherId=frmaster[0]}
  [177] = {x=12.816155, y=45.622354, z=113.994934, rx=0.000556, ry=-139.071531, rz=61.018527, shoulder=lefty, elbow=epositive, wrist=wpositive, fatherId=frmaster[0]}
  [178] = {x=8.99919, y=45.293989, z=114.519421, rx=0.000985, ry=-140.93465, rz=60.675039, shoulder=lefty, elbow=epositive, wrist=wpositive, fatherId=frmaster[0]}
  [179] = {x=5.229614, y=44.883576, z=114.94756, rx=0.001161, ry=-142.73729, rz=60.256643, shoulder=lefty, elbow=epositive, wrist=wpositive, fatherId=frmaster[0]}
  [180] = {x=1.451225, y=44.425237, z=115.26707, rx=-0.000034, ry=-144.523632, rz=59.799584, shoulder=lefty, elbow=epositive, wrist=wpositive, fatherId=frmaster[0]}
  [181] = {x=-2.307811, y=43.925262, z=115.471626, rx=0.001142, ry=-146.286475, rz=59.304388, shoulder=lefty, elbow=epositive, wrist=wpositive, fatherId=frmaster[0]}
  [182] = {x=-6.055853, y=43.371193, z=115.561954, rx=0.000111, ry=-148.020084, rz=58.766409, shoulder=lefty, elbow=epositive, wrist=wpositive, fatherId=frmaster[0]}
  [183] = {x=-9.712351, y=42.742693, z=115.565714, rx=-0.00009, ry=-149.688718, rz=58.161849, shoulder=lefty, elbow=epositive, wrist=wpositive, fatherId=frmaster[0]}
  [184] = {x=-13.323835, y=42.072162, z=115.469914, rx=-0.000531, ry=-151.324603, rz=57.526735, shoulder=lefty, elbow=epositive, wrist=wpositive, fatherId=frmaster[0]}
  [185] = {x=-16.86003, y=41.366653, z=115.277948, rx=0.000022, ry=-152.915853, rz=56.86152, shoulder=lefty, elbow=epositive, wrist=wpositive, fatherId=frmaster[0]}
  [186] = {x=-20.297697, y=40.619044, z=115.005604, rx=0.000334, ry=-154.453541, rz=56.166082, shoulder=lefty, elbow=epositive, wrist=wpositive, fatherId=frmaster[0]}
  [187] = {x=-26.789557, y=38.993633, z=114.245437, rx=-0.000366, ry=-157.317863, rz=54.675613, shoulder=lefty, elbow=epositive, wrist=wpositive, fatherId=frmaster[0]}
  [188] = {x=-32.775618, y=37.209323, z=113.281593, rx=-0.000484, ry=-159.921028, rz=53.068148, shoulder=lefty, elbow=epositive, wrist=wpositive, fatherId=frmaster[0]}
  [189] = {x=-38.202922, y=35.258076, z=112.197188, rx=0.000079, ry=-162.242584, rz=51.338647, shoulder=lefty, elbow=epositive, wrist=wpositive, fatherId=frmaster[0]}
  [190] = {x=-43.069992, y=33.141215, z=111.069429, rx=0.000738, ry=-164.287092, rz=49.495346, shoulder=lefty, elbow=epositive, wrist=wpositive, fatherId=frmaster[0]}
  [191] = {x=-47.48842, y=30.826973, z=109.908643, rx=0.000268, ry=-166.108815, rz=47.517105, shoulder=lefty, elbow=epositive, wrist=wpositive, fatherId=frmaster[0]}
  [192] = {x=-51.457313, y=28.300184, z=108.774635, rx=0.000767, ry=-167.714658, rz=45.388827, shoulder=lefty, elbow=epositive, wrist=wpositive, fatherId=frmaster[0]}
  [193] = {x=-58.259306, y=22.435274, z=106.621307, rx=-0.000006, ry=-170.380497, rz=40.578435, shoulder=lefty, elbow=epositive, wrist=wpositive, fatherId=frmaster[0]}
  [194] = {x=-63.469827, y=15.638668, z=104.756105, rx=-0.000224, ry=-172.388364, rz=35.154164, shoulder=lefty, elbow=epositive, wrist=wpositive, fatherId=frmaster[0]}
  [195] = {x=-69.233917, y=4.126795, z=101.950198, rx=0.000187, ry=-174.960019, rz=25.998384, shoulder=lefty, elbow=epositive, wrist=wpositive, fatherId=frmaster[0]}
  [196] = {x=-69.232978, y=4.123883, z=111.947011, rx=-0.001254, ry=-174.9603, rz=25.997917, shoulder=lefty, elbow=epositive, wrist=wpositive, fatherId=frmaster[0]}
  [197] = {x=-67.948878, y=4.126484, z=126.461204, rx=0.000749, ry=-174.960312, rz=25.998347, shoulder=lefty, elbow=epositive, wrist=wpositive, fatherId=frmaster[0]}
  [198] = {x=-68.941187, y=-2.594666, z=125.851852, rx=-179.999968, ry=-4.538961, rz=20.573522, shoulder=lefty, elbow=epositive, wrist=wpositive, fatherId=frmaster[0]}
  [199] = {x=-70.091269, y=-2.592516, z=111.352514, rx=-179.999154, ry=-4.538889, rz=20.573541, shoulder=lefty, elbow=epositive, wrist=wpositive, fatherId=frmaster[0]}
  [200] = {x=-70.091245, y=-2.592615, z=101.352, rx=-179.999967, ry=-4.539167, rz=20.573205, shoulder=lefty, elbow=epositive, wrist=wpositive, fatherId=frmaster[0]}
  [201] = {x=-65.560701, y=-4.52076, z=104.634327, rx=179.999719, ry=-7.320437, rz=18.95207, shoulder=lefty, elbow=epositive, wrist=wpositive, fatherId=frmaster[0]}
  [202] = {x=-62.144277, y=-5.717504, z=106.803129, rx=179.999641, ry=-9.281351, rz=17.978978, shoulder=lefty, elbow=epositive, wrist=wpositive, fatherId=frmaster[0]}
  [203] = {x=-57.806655, y=-7.017721, z=109.289468, rx=179.999337, ry=-11.675241, rz=16.938409, shoulder=lefty, elbow=epositive, wrist=wpositive, fatherId=frmaster[0]}
  [204] = {x=-55.21076, y=-7.694538, z=110.650126, rx=179.999593, ry=-13.066085, rz=16.401878, shoulder=lefty, elbow=epositive, wrist=wpositive, fatherId=frmaster[0]}
  [205] = {x=-52.128732, y=-8.432815, z=112.151089, rx=-179.999381, ry=-14.684501, rz=15.82104, shoulder=lefty, elbow=epositive, wrist=wpositive, fatherId=frmaster[0]}
  [206] = {x=-48.562509, y=-9.195661, z=113.731399, rx=179.999511, ry=-16.519177, rz=15.226365, shoulder=lefty, elbow=epositive, wrist=wpositive, fatherId=frmaster[0]}
  [207] = {x=-44.445238, y=-9.974206, z=115.393252, rx=-179.999681, ry=-18.599864, rz=14.620936, shoulder=lefty, elbow=epositive, wrist=wpositive, fatherId=frmaster[0]}
  [208] = {x=-39.805042, y=-10.739339, z=117.051018, rx=179.999427, ry=-20.909147, rz=14.030338, shoulder=lefty, elbow=epositive, wrist=wpositive, fatherId=frmaster[0]}
  [209] = {x=-34.571504, y=-11.488063, z=118.672785, rx=-179.999103, ry=-23.469203, rz=13.448615, shoulder=lefty, elbow=epositive, wrist=wpositive, fatherId=frmaster[0]}
  [210] = {x=-28.796804, y=-12.205792, z=120.171192, rx=-179.999925, ry=-26.258738, rz=12.893974, shoulder=lefty, elbow=epositive, wrist=wpositive, fatherId=frmaster[0]}
  [211] = {x=-25.705389, y=-12.553736, z=120.842951, rx=-179.999916, ry=-27.739104, rz=12.626325, shoulder=lefty, elbow=epositive, wrist=wpositive, fatherId=frmaster[0]}
  [212] = {x=-22.482081, y=-12.893063, z=121.465163, rx=-179.999286, ry=-29.2735, rz=12.362432, shoulder=lefty, elbow=epositive, wrist=wpositive, fatherId=frmaster[0]}
  [213] = {x=-19.099649, y=-13.220159, z=122.01174, rx=-179.999926, ry=-30.87363, rz=12.11146, shoulder=lefty, elbow=epositive, wrist=wpositive, fatherId=frmaster[0]}
  [214] = {x=-15.563891, y=-13.544095, z=122.485202, rx=179.999303, ry=-32.542436, rz=11.862282, shoulder=lefty, elbow=epositive, wrist=wpositive, fatherId=frmaster[0]}
  [215] = {x=-11.860292, y=-13.859789, z=122.869811, rx=179.999657, ry=-34.28039, rz=11.617688, shoulder=lefty, elbow=epositive, wrist=wpositive, fatherId=frmaster[0]}
  [216] = {x=-7.999201, y=-14.170821, z=123.152049, rx=-179.9993, ry=-36.089153, rz=11.376413, shoulder=lefty, elbow=epositive, wrist=wpositive, fatherId=frmaster[0]}
  [217] = {x=-3.976731, y=-14.469679, z=123.320363, rx=-179.998203, ry=-37.973408, rz=11.147405, shoulder=lefty, elbow=epositive, wrist=wpositive, fatherId=frmaster[0]}
  [218] = {x=-0.001611, y=-14.755184, z=123.349313, rx=-179.999213, ry=-39.835789, rz=10.926322, shoulder=lefty, elbow=epositive, wrist=wpositive, fatherId=frmaster[0]}
  [219] = {x=3.921658, y=-15.027909, z=123.245131, rx=179.999493, ry=-41.674416, rz=10.717247, shoulder=lefty, elbow=epositive, wrist=wpositive, fatherId=frmaster[0]}
  [220] = {x=7.787656, y=-15.282792, z=123.030151, rx=-179.998199, ry=-43.486, rz=10.518616, shoulder=lefty, elbow=epositive, wrist=wpositive, fatherId=frmaster[0]}
  [221] = {x=3.632632, y=-13.0539, z=123.518074, rx=179.99995, ry=-41.686437, rz=12.370731, shoulder=lefty, elbow=epositive, wrist=wpositive, fatherId=frmaster[0]}
  [222] = {x=-0.116628, y=-10.553936, z=123.837966, rx=-179.999968, ry=-40.072424, rz=14.411441, shoulder=lefty, elbow=epositive, wrist=wpositive, fatherId=frmaster[0]}
  [223] = {x=-2.870576, y=-7.779605, z=124.040599, rx=-179.999105, ry=-38.909745, rz=16.640287, shoulder=lefty, elbow=epositive, wrist=wpositive, fatherId=frmaster[0]}
  [224] = {x=-5.004213, y=-4.719529, z=124.142877, rx=-179.998694, ry=-38.009932, rz=19.065288, shoulder=lefty, elbow=epositive, wrist=wpositive, fatherId=frmaster[0]}
  [225] = {x=-6.286234, y=-1.405857, z=124.170085, rx=-179.999075, ry=-37.465546, rz=21.665507, shoulder=lefty, elbow=epositive, wrist=wpositive, fatherId=frmaster[0]}
  [226] = {x=-6.763491, y=1.995044, z=124.139406, rx=-179.999796, ry=-37.246434, rz=24.324557, shoulder=lefty, elbow=epositive, wrist=wpositive, fatherId=frmaster[0]}
  [227] = {x=-6.628353, y=5.404754, z=124.035693, rx=179.999483, ry=-37.250746, rz=26.994765, shoulder=lefty, elbow=epositive, wrist=wpositive, fatherId=frmaster[0]}
  [228] = {x=-5.669968, y=8.784748, z=123.870598, rx=-179.999027, ry=-37.580312, rz=29.65073, shoulder=lefty, elbow=epositive, wrist=wpositive, fatherId=frmaster[0]}
  [229] = {x=-4.462138, y=12.188846, z=123.600895, rx=179.999877, ry=-37.973856, rz=32.334503, shoulder=lefty, elbow=epositive, wrist=wpositive, fatherId=frmaster[0]}
  [230] = {x=-2.489646, y=15.635578, z=123.227559, rx=179.998826, ry=-38.667471, rz=35.069591, shoulder=lefty, elbow=epositive, wrist=wpositive, fatherId=frmaster[0]}
  [231] = {x=-0.697365, y=19.173794, z=122.703604, rx=179.999639, ry=-39.205656, rz=37.895465, shoulder=lefty, elbow=epositive, wrist=wpositive, fatherId=frmaster[0]}
  [232] = {x=1.761902, y=22.681657, z=122.038748, rx=-179.999829, ry=-40.003178, rz=40.733105, shoulder=lefty, elbow=epositive, wrist=wpositive, fatherId=frmaster[0]}
  [233] = {x=3.610937, y=26.090403, z=121.250151, rx=-179.999942, ry=-40.461127, rz=43.535028, shoulder=lefty, elbow=epositive, wrist=wpositive, fatherId=frmaster[0]}
  [234] = {x=6.005086, y=29.344743, z=120.329381, rx=-179.999476, ry=-41.144604, rz=46.265313, shoulder=lefty, elbow=epositive, wrist=wpositive, fatherId=frmaster[0]}
  [235] = {x=8.175238, y=32.513013, z=119.28988, rx=179.999815, ry=-41.674279, rz=48.981987, shoulder=lefty, elbow=epositive, wrist=wpositive, fatherId=frmaster[0]}
  [236] = {x=10.804669, y=35.563809, z=118.108795, rx=-179.999695, ry=-42.396993, rz=51.657982, shoulder=lefty, elbow=epositive, wrist=wpositive, fatherId=frmaster[0]}
  [237] = {x=13.537862, y=38.530039, z=116.77667, rx=179.999723, ry=-43.14025, rz=54.327489, shoulder=lefty, elbow=epositive, wrist=wpositive, fatherId=frmaster[0]}
  [238] = {x=16.594305, y=41.382503, z=115.269063, rx=-179.999776, ry=-44.022413, rz=56.970299, shoulder=lefty, elbow=epositive, wrist=wpositive, fatherId=frmaster[0]}
  [239] = {x=19.918306, y=44.041072, z=113.61946, rx=-179.999049, ry=-45.050182, rz=59.514719, shoulder=lefty, elbow=epositive, wrist=wpositive, fatherId=frmaster[0]}
  [240] = {x=23.334897, y=46.459403, z=111.834207, rx=179.998974, ry=-46.157591, rz=61.920851, shoulder=lefty, elbow=epositive, wrist=wpositive, fatherId=frmaster[0]}
  [241] = {x=19.980834, y=46.20086, z=112.638726, rx=179.999942, ry=-44.473108, rz=61.638901, shoulder=lefty, elbow=epositive, wrist=wpositive, fatherId=frmaster[0]}
  [242] = {x=16.481484, y=45.924464, z=113.358772, rx=-179.999155, ry=-42.731493, rz=61.33928, shoulder=lefty, elbow=epositive, wrist=wpositive, fatherId=frmaster[0]}
  [243] = {x=12.816155, y=45.622354, z=113.994934, rx=-179.999444, ry=-40.928469, rz=61.018527, shoulder=lefty, elbow=epositive, wrist=wpositive, fatherId=frmaster[0]}
  [244] = {x=8.99919, y=45.293989, z=114.519421, rx=-179.999015, ry=-39.06535, rz=60.675039, shoulder=lefty, elbow=epositive, wrist=wpositive, fatherId=frmaster[0]}
  [245] = {x=5.229614, y=44.883576, z=114.94756, rx=-179.998839, ry=-37.26271, rz=60.256643, shoulder=lefty, elbow=epositive, wrist=wpositive, fatherId=frmaster[0]}
  [246] = {x=1.451225, y=44.425237, z=115.26707, rx=179.999966, ry=-35.476368, rz=59.799584, shoulder=lefty, elbow=epositive, wrist=wpositive, fatherId=frmaster[0]}
  [247] = {x=-2.307811, y=43.925262, z=115.471626, rx=-179.998858, ry=-33.713525, rz=59.304388, shoulder=lefty, elbow=epositive, wrist=wpositive, fatherId=frmaster[0]}
  [248] = {x=-6.055853, y=43.371193, z=115.561954, rx=-179.999889, ry=-31.979916, rz=58.766409, shoulder=lefty, elbow=epositive, wrist=wpositive, fatherId=frmaster[0]}
  [249] = {x=-9.712351, y=42.742693, z=115.565714, rx=179.99991, ry=-30.311282, rz=58.161849, shoulder=lefty, elbow=epositive, wrist=wpositive, fatherId=frmaster[0]}
  [250] = {x=-13.323835, y=42.072162, z=115.469914, rx=179.999469, ry=-28.675397, rz=57.526735, shoulder=lefty, elbow=epositive, wrist=wpositive, fatherId=frmaster[0]}
  [251] = {x=-16.86003, y=41.366653, z=115.277948, rx=-179.999978, ry=-27.084147, rz=56.86152, shoulder=lefty, elbow=epositive, wrist=wpositive, fatherId=frmaster[0]}
  [252] = {x=-20.297697, y=40.619044, z=115.005604, rx=-179.999666, ry=-25.546459, rz=56.166082, shoulder=lefty, elbow=epositive, wrist=wpositive, fatherId=frmaster[0]}
  [253] = {x=-26.789557, y=38.993633, z=114.245437, rx=179.999634, ry=-22.682137, rz=54.675613, shoulder=lefty, elbow=epositive, wrist=wpositive, fatherId=frmaster[0]}
  [254] = {x=-32.775618, y=37.209323, z=113.281593, rx=179.999516, ry=-20.078972, rz=53.068148, shoulder=lefty, elbow=epositive, wrist=wpositive, fatherId=frmaster[0]}
  [255] = {x=-38.202922, y=35.258076, z=112.197188, rx=-179.999921, ry=-17.757416, rz=51.338647, shoulder=lefty, elbow=epositive, wrist=wpositive, fatherId=frmaster[0]}
  [256] = {x=-43.069992, y=33.141215, z=111.069429, rx=-179.999262, ry=-15.712908, rz=49.495346, shoulder=lefty, elbow=epositive, wrist=wpositive, fatherId=frmaster[0]}
  [257] = {x=-47.48842, y=30.826973, z=109.908643, rx=-179.999732, ry=-13.891185, rz=47.517105, shoulder=lefty, elbow=epositive, wrist=wpositive, fatherId=frmaster[0]}
  [258] = {x=-51.457313, y=28.300184, z=108.774635, rx=-179.999233, ry=-12.285342, rz=45.388827, shoulder=lefty, elbow=epositive, wrist=wpositive, fatherId=frmaster[0]}
  [259] = {x=-58.259306, y=22.435274, z=106.621307, rx=179.999994, ry=-9.619503, rz=40.578435, shoulder=lefty, elbow=epositive, wrist=wpositive, fatherId=frmaster[0]}
  [260] = {x=-63.469827, y=15.638668, z=104.756105, rx=179.999776, ry=-7.611636, rz=35.154164, shoulder=lefty, elbow=epositive, wrist=wpositive, fatherId=frmaster[0]}
  [261] = {x=-69.233917, y=4.126795, z=101.950198, rx=-179.999813, ry=-5.039981, rz=25.998384, shoulder=lefty, elbow=epositive, wrist=wpositive, fatherId=frmaster[0]}
  [262] = {x=-69.232978, y=4.123883, z=111.947011, rx=179.998746, ry=-5.0397, rz=25.997917, shoulder=lefty, elbow=epositive, wrist=wpositive, fatherId=frmaster[0]}
pointRx pdemo1[713]
  [0] = {x=-18.96517, y=-20.048024, z=152.6932, rx=-0.000601, ry=-174.211459, rz=89.999998, shoulder=lefty, elbow=epositive, wrist=wpositive, fatherId=frmaster[1]}
  [1] = {x=-23.462584, y=-20.043665, z=108.32512, rx=-179.999883, ry=-5.787827, rz=-89.99982, shoulder=lefty, elbow=epositive, wrist=wpositive, fatherId=frmaster[1]}
  [2] = {x=-23.463232, y=-20.044107, z=98.317618, rx=-179.999811, ry=-5.787538, rz=-89.999354, shoulder=lefty, elbow=epositive, wrist=wpositive, fatherId=frmaster[1]}
  [3] = {x=-19.816641, y=-20.425168, z=99.208339, rx=179.999752, ry=-8.130371, rz=-89.999727, shoulder=lefty, elbow=epositive, wrist=wpositive, fatherId=frmaster[1]}
  [4] = {x=-15.087203, y=-20.853749, z=100.100863, rx=179.999972, ry=-11.043087, rz=-89.999026, shoulder=lefty, elbow=epositive, wrist=wpositive, fatherId=frmaster[1]}
  [5] = {x=-10.366022, y=-21.350672, z=100.726684, rx=-0.000315, ry=-166.115847, rz=89.999913, shoulder=lefty, elbow=epositive, wrist=wpositive, fatherId=frmaster[1]}
  [6] = {x=-7.645382, y=-21.597594, z=100.981381, rx=-0.00024, ry=-164.497107, rz=89.999759, shoulder=lefty, elbow=epositive, wrist=wpositive, fatherId=frmaster[1]}
  [7] = {x=-4.684522, y=-21.841423, z=101.168911, rx=-179.999911, ry=-17.255988, rz=-89.999902, shoulder=lefty, elbow=epositive, wrist=wpositive, fatherId=frmaster[1]}
  [8] = {x=0.189055, y=-22.373885, z=101.279298, rx=-179.999692, ry=-20.123277, rz=-89.99962, shoulder=lefty, elbow=epositive, wrist=wpositive, fatherId=frmaster[1]}
  [9] = {x=2.844715, y=-22.644904, z=101.243444, rx=0.0003, ry=-158.320767, rz=89.999914, shoulder=lefty, elbow=epositive, wrist=wpositive, fatherId=frmaster[1]}
  [10] = {x=5.634284, y=-22.915698, z=101.1174, rx=0.000418, ry=-156.686411, rz=89.999139, shoulder=lefty, elbow=epositive, wrist=wpositive, fatherId=frmaster[1]}
  [11] = {x=10.528438, y=-23.452167, z=100.715388, rx=179.999768, ry=-26.184957, rz=-89.999583, shoulder=lefty, elbow=epositive, wrist=wpositive, fatherId=frmaster[1]}
  [12] = {x=13.642756, y=-23.993218, z=100.326624, rx=-179.999809, ry=-28.051053, rz=-89.999357, shoulder=lefty, elbow=epositive, wrist=wpositive, fatherId=frmaster[1]}
  [13] = {x=16.483896, y=-24.55078, z=99.874232, rx=-0.000517, ry=-150.237765, rz=89.998988, shoulder=lefty, elbow=epositive, wrist=wpositive, fatherId=frmaster[1]}
  [14] = {x=19.255095, y=-25.101295, z=99.349236, rx=0.000098, ry=-148.559215, rz=89.999065, shoulder=lefty, elbow=epositive, wrist=wpositive, fatherId=frmaster[1]}
  [15] = {x=21.951218, y=-25.651654, z=98.756801, rx=-0.000182, ry=-146.91019, rz=89.999619, shoulder=lefty, elbow=epositive, wrist=wpositive, fatherId=frmaster[1]}
  [16] = {x=24.579683, y=-26.199417, z=98.09306, rx=-179.999575, ry=-34.707902, rz=-89.999357, shoulder=lefty, elbow=epositive, wrist=wpositive, fatherId=frmaster[1]}
  [17] = {x=29.278158, y=-27.315982, z=96.72306, rx=-0.000524, ry=-142.365013, rz=89.998933, shoulder=lefty, elbow=epositive, wrist=wpositive, fatherId=frmaster[1]}
  [18] = {x=33.815844, y=-28.426565, z=95.143172, rx=-0.000545, ry=-139.490786, rz=89.999611, shoulder=lefty, elbow=epositive, wrist=wpositive, fatherId=frmaster[1]}
  [19] = {x=37.993518, y=-29.533967, z=93.448805, rx=-179.999232, ry=-43.210814, rz=-89.998713, shoulder=lefty, elbow=epositive, wrist=wpositive, fatherId=frmaster[1]}
  [20] = {x=40.334597, y=-30.09312, z=92.400878, rx=-0.000153, ry=-135.266825, rz=89.999997, shoulder=lefty, elbow=epositive, wrist=wpositive, fatherId=frmaster[1]}
  [21] = {x=43.092152, y=-30.650175, z=91.093242, rx=-179.999714, ry=-46.53747, rz=-89.99916, shoulder=lefty, elbow=epositive, wrist=wpositive, fatherId=frmaster[1]}
  [22] = {x=45.946869, y=-31.210457, z=89.624058, rx=-0.000667, ry=-131.572098, rz=89.999114, shoulder=lefty, elbow=epositive, wrist=wpositive, fatherId=frmaster[1]}
  [23] = {x=49.020952, y=-31.768062, z=87.910405, rx=-0.000712, ry=-129.504767, rz=89.999679, shoulder=lefty, elbow=epositive, wrist=wpositive, fatherId=frmaster[1]}
  [24] = {x=52.333983, y=-32.326895, z=85.907964, rx=-0.000763, ry=-127.235317, rz=89.999387, shoulder=lefty, elbow=epositive, wrist=wpositive, fatherId=frmaster[1]}
  [25] = {x=55.895707, y=-32.881512, z=83.548498, rx=-179.999162, ry=-55.258831, rz=-89.999513, shoulder=lefty, elbow=epositive, wrist=wpositive, fatherId=frmaster[1]}
  [26] = {x=59.512133, y=-33.441317, z=80.922892, rx=0.000599, ry=-122.139441, rz=89.999688, shoulder=lefty, elbow=epositive, wrist=wpositive, fatherId=frmaster[1]}
  [27] = {x=63.397094, y=-34.00372, z=77.822685, rx=-179.999865, ry=-60.751412, rz=-89.999836, shoulder=lefty, elbow=epositive, wrist=wpositive, fatherId=frmaster[1]}
  [28] = {x=65.432612, y=-34.285528, z=76.074093, rx=-0.001714, ry=-117.686829, rz=89.998746, shoulder=lefty, elbow=epositive, wrist=wpositive, fatherId=frmaster[1]}
  [29] = {x=67.520447, y=-34.557953, z=74.164172, rx=-179.999023, ry=-63.953784, rz=-89.998838, shoulder=lefty, elbow=epositive, wrist=wpositive, fatherId=frmaster[1]}
  [30] = {x=69.660663, y=-34.838665, z=72.104425, rx=-179.998935, ry=-65.675779, rz=-89.999167, shoulder=lefty, elbow=epositive, wrist=wpositive, fatherId=frmaster[1]}
  [31] = {x=71.834063, y=-35.120891, z=69.874135, rx=-0.000593, ry=-112.523327, rz=89.998808, shoulder=lefty, elbow=epositive, wrist=wpositive, fatherId=frmaster[1]}
  [32] = {x=73.952222, y=-35.400144, z=67.567091, rx=0.00012, ry=-110.706298, rz=89.999449, shoulder=lefty, elbow=epositive, wrist=wpositive, fatherId=frmaster[1]}
  [33] = {x=76.112362, y=-35.678593, z=65.05668, rx=-179.998546, ry=-71.210166, rz=-89.998874, shoulder=lefty, elbow=epositive, wrist=wpositive, fatherId=frmaster[1]}
  [34] = {x=78.296393, y=-35.963382, z=62.344514, rx=-0.001071, ry=-106.772201, rz=89.999015, shoulder=lefty, elbow=epositive, wrist=wpositive, fatherId=frmaster[1]}
  [35] = {x=80.486593, y=-36.242456, z=59.412826, rx=-0.001948, ry=-104.659789, rz=89.99825, shoulder=lefty, elbow=epositive, wrist=wpositive, fatherId=frmaster[1]}
  [36] = {x=82.649534, y=-36.51962, z=56.27084, rx=-0.000501, ry=-102.455387, rz=89.999177, shoulder=lefty, elbow=epositive, wrist=wpositive, fatherId=frmaster[1]}
  [37] = {x=84.766181, y=-36.800484, z=52.938193, rx=-0.001841, ry=-100.1706, rz=89.998114, shoulder=lefty, elbow=epositive, wrist=wpositive, fatherId=frmaster[1]}
  [38] = {x=86.814683, y=-37.081591, z=49.408559, rx=-0.005376, ry=-97.819747, rz=89.994372, shoulder=lefty, elbow=epositive, wrist=wpositive, fatherId=frmaster[1]}
  [39] = {x=88.824909, y=-37.358634, z=45.578394, rx=-0.00118, ry=-95.317641, rz=89.998858, shoulder=lefty, elbow=epositive, wrist=wpositive, fatherId=frmaster[1]}
  [40] = {x=90.050848, y=-37.497721, z=43.043255, rx=-0.00116, ry=-93.69812, rz=89.998427, shoulder=lefty, elbow=epositive, wrist=wpositive, fatherId=frmaster[1]}
  [41] = {x=91.127073, y=-37.63701, z=40.649221, rx=-179.997932, ry=-87.821738, rz=-89.998136, shoulder=lefty, elbow=epositive, wrist=wpositive, fatherId=frmaster[1]}
  [42] = {x=92.886481, y=-37.917172, z=36.297912, rx=-0.038358, ry=-89.473525, rz=89.961729, shoulder=lefty, elbow=epositive, wrist=wpositive, fatherId=frmaster[1]}
  [43] = {x=94.169327, y=-38.197827, z=32.647914, rx=-0.007009, ry=-87.235981, rz=89.992919, shoulder=lefty, elbow=epositive, wrist=wpositive, fatherId=frmaster[1]}
  [44] = {x=95.072423, y=-38.481114, z=29.737512, rx=0.005732, ry=-85.470452, rz=90.005704, shoulder=lefty, elbow=epositive, wrist=wpositive, fatherId=frmaster[1]}
  [45] = {x=96.062811, y=-39.595291, z=25.468303, rx=-0.005344, ry=-82.913438, rz=89.994551, shoulder=lefty, elbow=epositive, wrist=wpositive, fatherId=frmaster[1]}
  [46] = {x=96.046175, y=-41.825416, z=23.544635, rx=-0.00046, ry=-81.767404, rz=89.998969, shoulder=lefty, elbow=epositive, wrist=wpositive, fatherId=frmaster[1]}
  [47] = {x=96.266015, y=-44.047585, z=20.151312, rx=0.003085, ry=-79.748331, rz=90.002429, shoulder=lefty, elbow=epositive, wrist=wpositive, fatherId=frmaster[1]}
  [48] = {x=95.837317, y=-46.263529, z=19.527719, rx=-0.002879, ry=-79.374252, rz=89.997297, shoulder=lefty, elbow=epositive, wrist=wpositive, fatherId=frmaster[1]}
  [49] = {x=95.228564, y=-48.470385, z=19.531167, rx=0.000601, ry=-79.373755, rz=90.000801, shoulder=lefty, elbow=epositive, wrist=wpositive, fatherId=frmaster[1]}
  [50] = {x=94.621665, y=-50.681168, z=19.529466, rx=0.004255, ry=-79.373694, rz=90.004145, shoulder=lefty, elbow=epositive, wrist=wpositive, fatherId=frmaster[1]}
  [51] = {x=93.95764, y=-52.870174, z=19.527425, rx=0.002544, ry=-79.373361, rz=90.002577, shoulder=lefty, elbow=epositive, wrist=wpositive, fatherId=frmaster[1]}
  [52] = {x=93.290826, y=-55.055756, z=19.5317, rx=-0.002571, ry=-79.37359, rz=89.997804, shoulder=lefty, elbow=epositive, wrist=wpositive, fatherId=frmaster[1]}
  [53] = {x=92.578024, y=-57.230281, z=19.527844, rx=-0.001394, ry=-79.374147, rz=89.998226, shoulder=lefty, elbow=epositive, wrist=wpositive, fatherId=frmaster[1]}
  [54] = {x=91.860552, y=-59.403243, z=19.527909, rx=-0.00089, ry=-79.373882, rz=89.998842, shoulder=lefty, elbow=epositive, wrist=wpositive, fatherId=frmaster[1]}
  [55] = {x=91.095542, y=-61.56469, z=19.526877, rx=0.003026, ry=-79.374406, rz=90.002721, shoulder=lefty, elbow=epositive, wrist=wpositive, fatherId=frmaster[1]}
  [56] = {x=90.320474, y=-63.717023, z=19.531145, rx=-0.001214, ry=-79.373131, rz=89.999229, shoulder=lefty, elbow=epositive, wrist=wpositive, fatherId=frmaster[1]}
  [57] = {x=91.228747, y=-61.66316, z=19.526312, rx=0.000084, ry=-79.37396, rz=90.000189, shoulder=lefty, elbow=epositive, wrist=wpositive, fatherId=frmaster[1]}
  [58] = {x=92.127797, y=-59.609161, z=19.53008, rx=0.000133, ry=-79.372968, rz=90.000323, shoulder=lefty, elbow=epositive, wrist=wpositive, fatherId=frmaster[1]}
  [59] = {x=93.028542, y=-57.554175, z=19.53221, rx=-0.001578, ry=-79.373323, rz=89.998477, shoulder=lefty, elbow=epositive, wrist=wpositive, fatherId=frmaster[1]}
  [60] = {x=93.662663, y=-55.991824, z=19.52775, rx=-0.001468, ry=-79.374224, rz=89.998285, shoulder=lefty, elbow=epositive, wrist=wpositive, fatherId=frmaster[1]}
  [61] = {x=94.296939, y=-54.43705, z=19.529438, rx=0.000918, ry=-79.374154, rz=90.00127, shoulder=lefty, elbow=epositive, wrist=wpositive, fatherId=frmaster[1]}
  [62] = {x=94.863447, y=-52.851806, z=19.525072, rx=-0.002321, ry=-79.374373, rz=89.997391, shoulder=lefty, elbow=epositive, wrist=wpositive, fatherId=frmaster[1]}
  [63] = {x=95.432367, y=-51.273675, z=19.531293, rx=0.001414, ry=-79.373279, rz=90.001068, shoulder=lefty, elbow=epositive, wrist=wpositive, fatherId=frmaster[1]}
  [64] = {x=95.912547, y=-49.676085, z=19.525984, rx=0.000698, ry=-79.374074, rz=89.999925, shoulder=lefty, elbow=epositive, wrist=wpositive, fatherId=frmaster[1]}
  [65] = {x=96.266507, y=-48.081467, z=20.132369, rx=0.000274, ry=-79.732044, rz=89.999839, shoulder=lefty, elbow=epositive, wrist=wpositive, fatherId=frmaster[1]}
  [66] = {x=96.133261, y=-46.456619, z=22.368479, rx=-0.002438, ry=-81.061483, rz=89.998538, shoulder=lefty, elbow=epositive, wrist=wpositive, fatherId=frmaster[1]}
  [67] = {x=95.955405, y=-44.830171, z=24.588227, rx=0.001748, ry=-82.390629, rz=90.000856, shoulder=lefty, elbow=epositive, wrist=wpositive, fatherId=frmaster[1]}
  [68] = {x=95.79268, y=-43.182447, z=26.201876, rx=0.005028, ry=-83.35179, rz=90.0051, shoulder=lefty, elbow=epositive, wrist=wpositive, fatherId=frmaster[1]}
  [69] = {x=96.045158, y=-41.517917, z=25.928219, rx=-0.007242, ry=-83.190708, rz=89.992907, shoulder=lefty, elbow=epositive, wrist=wpositive, fatherId=frmaster[1]}
  [70] = {x=95.482935, y=-39.856574, z=28.2622, rx=0.000769, ry=-84.586254, rz=90.000254, shoulder=lefty, elbow=epositive, wrist=wpositive, fatherId=frmaster[1]}
  [71] = {x=95.459578, y=-38.189355, z=28.340385, rx=0.0023, ry=-84.630238, rz=90.002356, shoulder=lefty, elbow=epositive, wrist=wpositive, fatherId=frmaster[1]}
  [72] = {x=96.037569, y=-36.527529, z=25.982306, rx=0.002157, ry=-83.22462, rz=90.002085, shoulder=lefty, elbow=epositive, wrist=wpositive, fatherId=frmaster[1]}
  [73] = {x=95.794712, y=-34.877576, z=26.179177, rx=0.003564, ry=-83.33604, rz=90.004018, shoulder=lefty, elbow=epositive, wrist=wpositive, fatherId=frmaster[1]}
  [74] = {x=96.064268, y=-32.418334, z=23.259632, rx=-0.005638, ry=-81.595045, rz=89.994441, shoulder=lefty, elbow=epositive, wrist=wpositive, fatherId=frmaster[1]}
  [75] = {x=96.263652, y=-30.612383, z=20.193509, rx=0.003461, ry=-79.771799, rz=90.002604, shoulder=lefty, elbow=epositive, wrist=wpositive, fatherId=frmaster[1]}
  [76] = {x=95.49089, y=-27.953041, z=19.530394, rx=0.001426, ry=-79.373507, rz=90.001737, shoulder=lefty, elbow=epositive, wrist=wpositive, fatherId=frmaster[1]}
  [77] = {x=94.434398, y=-25.344644, z=19.530202, rx=-0.000192, ry=-79.373477, rz=89.99986, shoulder=lefty, elbow=epositive, wrist=wpositive, fatherId=frmaster[1]}
  [78] = {x=93.749368, y=-23.815417, z=19.526527, rx=0.000499, ry=-79.373989, rz=89.999983, shoulder=lefty, elbow=epositive, wrist=wpositive, fatherId=frmaster[1]}
  [79] = {x=93.062244, y=-22.293387, z=19.533582, rx=-0.000205, ry=-79.373016, rz=89.999831, shoulder=lefty, elbow=epositive, wrist=wpositive, fatherId=frmaster[1]}
  [80] = {x=91.992807, y=-20.011623, z=19.525869, rx=-0.000988, ry=-79.37419, rz=89.998491, shoulder=lefty, elbow=epositive, wrist=wpositive, fatherId=frmaster[1]}
  [81] = {x=90.922863, y=-17.733633, z=19.532639, rx=0.001258, ry=-79.373379, rz=90.001328, shoulder=lefty, elbow=epositive, wrist=wpositive, fatherId=frmaster[1]}
  [82] = {x=89.890725, y=-15.434378, z=19.528964, rx=-0.001531, ry=-79.373477, rz=89.998434, shoulder=lefty, elbow=epositive, wrist=wpositive, fatherId=frmaster[1]}
  [83] = {x=88.934538, y=-13.10297, z=19.528885, rx=-0.003317, ry=-79.373864, rz=89.996723, shoulder=lefty, elbow=epositive, wrist=wpositive, fatherId=frmaster[1]}
  [84] = {x=88.392361, y=-11.526994, z=19.531886, rx=-0.000966, ry=-79.373729, rz=89.998911, shoulder=lefty, elbow=epositive, wrist=wpositive, fatherId=frmaster[1]}
  [85] = {x=87.853757, y=-9.954341, z=19.526278, rx=0.002189, ry=-79.374419, rz=90.002179, shoulder=lefty, elbow=epositive, wrist=wpositive, fatherId=frmaster[1]}
  [86] = {x=87.415435, y=-8.342749, z=19.531441, rx=0.000584, ry=-79.373558, rz=90.000369, shoulder=lefty, elbow=epositive, wrist=wpositive, fatherId=frmaster[1]}
  [87] = {x=87.073406, y=-6.714559, z=19.532016, rx=-0.001715, ry=-79.372919, rz=89.999051, shoulder=lefty, elbow=epositive, wrist=wpositive, fatherId=frmaster[1]}
  [88] = {x=86.840974, y=-5.087755, z=19.526356, rx=0.003412, ry=-79.374095, rz=90.003341, shoulder=lefty, elbow=epositive, wrist=wpositive, fatherId=frmaster[1]}
  [89] = {x=86.725259, y=-3.445654, z=19.527354, rx=-0.000424, ry=-79.374397, rz=89.999682, shoulder=lefty, elbow=epositive, wrist=wpositive, fatherId=frmaster[1]}
  [90] = {x=86.740178, y=-1.797732, z=19.525044, rx=-0.002624, ry=-79.374444, rz=89.996754, shoulder=lefty, elbow=epositive, wrist=wpositive, fatherId=frmaster[1]}
  [91] = {x=86.896045, y=-0.153671, z=19.532037, rx=-0.004358, ry=-79.373087, rz=89.995942, shoulder=lefty, elbow=epositive, wrist=wpositive, fatherId=frmaster[1]}
  [92] = {x=87.166189, y=1.465785, z=19.528435, rx=-0.001803, ry=-79.373886, rz=89.998082, shoulder=lefty, elbow=epositive, wrist=wpositive, fatherId=frmaster[1]}
  [93] = {x=87.53369, y=3.066256, z=19.53121, rx=-0.003854, ry=-79.373133, rz=89.996635, shoulder=lefty, elbow=epositive, wrist=wpositive, fatherId=frmaster[1]}
  [94] = {x=87.98834, y=4.646579, z=19.528823, rx=0.001143, ry=-79.37397, rz=90.001418, shoulder=lefty, elbow=epositive, wrist=wpositive, fatherId=frmaster[1]}
  [95] = {x=88.512507, y=6.204742, z=19.529314, rx=-0.000445, ry=-79.373285, rz=89.999848, shoulder=lefty, elbow=epositive, wrist=wpositive, fatherId=frmaster[1]}
  [96] = {x=89.129542, y=7.74888, z=19.526506, rx=-0.000701, ry=-79.374221, rz=89.99953, shoulder=lefty, elbow=epositive, wrist=wpositive, fatherId=frmaster[1]}
  [97] = {x=89.747284, y=9.293228, z=19.530787, rx=-0.000397, ry=-79.37372, rz=89.999684, shoulder=lefty, elbow=epositive, wrist=wpositive, fatherId=frmaster[1]}
  [98] = {x=90.438941, y=10.810892, z=19.529618, rx=-0.00373, ry=-79.37359, rz=89.996175, shoulder=lefty, elbow=epositive, wrist=wpositive, fatherId=frmaster[1]}
  [99] = {x=91.128111, y=12.326224, z=19.529442, rx=-0.003213, ry=-79.373893, rz=89.997359, shoulder=lefty, elbow=epositive, wrist=wpositive, fatherId=frmaster[1]}
  [100] = {x=91.862245, y=13.84145, z=19.527886, rx=-0.000147, ry=-79.373624, rz=89.999882, shoulder=lefty, elbow=epositive, wrist=wpositive, fatherId=frmaster[1]}
  [101] = {x=92.58979, y=15.36052, z=19.52744, rx=0.0015, ry=-79.373792, rz=90.001754, shoulder=lefty, elbow=epositive, wrist=wpositive, fatherId=frmaster[1]}
  [102] = {x=93.647835, y=17.661437, z=19.529965, rx=-0.001835, ry=-79.374199, rz=89.998558, shoulder=lefty, elbow=epositive, wrist=wpositive, fatherId=frmaster[1]}
  [103] = {x=94.7088, y=19.960675, z=19.527591, rx=-0.000119, ry=-79.374439, rz=89.999275, shoulder=lefty, elbow=epositive, wrist=wpositive, fatherId=frmaster[1]}
  [104] = {x=95.652771, y=22.307799, z=19.525888, rx=-0.000566, ry=-79.374239, rz=89.999563, shoulder=lefty, elbow=epositive, wrist=wpositive, fatherId=frmaster[1]}
  [105] = {x=96.23447, y=24.68915, z=20.694909, rx=-0.001625, ry=-80.067666, rz=89.998419, shoulder=lefty, elbow=epositive, wrist=wpositive, fatherId=frmaster[1]}
  [106] = {x=96.04524, y=26.297139, z=23.561751, rx=0.00165, ry=-81.776061, rz=90.001376, shoulder=lefty, elbow=epositive, wrist=wpositive, fatherId=frmaster[1]}
  [107] = {x=95.816163, y=27.930511, z=25.96336, rx=0.002697, ry=-83.21058, rz=90.002758, shoulder=lefty, elbow=epositive, wrist=wpositive, fatherId=frmaster[1]}
  [108] = {x=95.557185, y=29.578708, z=27.9832, rx=0.002192, ry=-84.418373, rz=90.001815, shoulder=lefty, elbow=epositive, wrist=wpositive, fatherId=frmaster[1]}
  [109] = {x=94.176415, y=30.411075, z=32.629247, rx=-0.0037, ry=-87.221962, rz=89.995898, shoulder=lefty, elbow=epositive, wrist=wpositive, fatherId=frmaster[1]}
  [110] = {x=93.067377, y=30.823323, z=35.817489, rx=0.034891, ry=-89.172193, rz=90.035328, shoulder=lefty, elbow=epositive, wrist=wpositive, fatherId=frmaster[1]}
  [111] = {x=91.597633, y=31.242188, z=39.546393, rx=-0.003301, ry=-91.486065, rz=89.996808, shoulder=lefty, elbow=epositive, wrist=wpositive, fatherId=frmaster[1]}
  [112] = {x=90.577095, y=31.656721, z=41.897016, rx=-0.003888, ry=-92.967845, rz=89.996375, shoulder=lefty, elbow=epositive, wrist=wpositive, fatherId=frmaster[1]}
  [113] = {x=89.407817, y=32.076137, z=44.4026, rx=-0.0018, ry=-94.560839, rz=89.997643, shoulder=lefty, elbow=epositive, wrist=wpositive, fatherId=frmaster[1]}
  [114] = {x=87.1947, y=32.911792, z=48.708758, rx=-179.997777, ry=-82.644088, rz=-89.997375, shoulder=lefty, elbow=epositive, wrist=wpositive, fatherId=frmaster[1]}
  [115] = {x=85.835727, y=34.584226, z=51.139026, rx=179.999322, ry=-81.03865, rz=-89.999777, shoulder=lefty, elbow=epositive, wrist=wpositive, fatherId=frmaster[1]}
  [116] = {x=88.247139, y=36.262646, z=46.717086, rx=-179.994475, ry=-83.945048, rz=-89.994394, shoulder=lefty, elbow=epositive, wrist=wpositive, fatherId=frmaster[1]}
  [117] = {x=89.691321, y=37.094903, z=43.809563, rx=-0.006466, ry=-94.183858, rz=89.992847, shoulder=lefty, elbow=epositive, wrist=wpositive, fatherId=frmaster[1]}
  [118] = {x=91.026629, y=37.93181, z=40.883211, rx=-0.000259, ry=-92.324634, rz=89.999824, shoulder=lefty, elbow=epositive, wrist=wpositive, fatherId=frmaster[1]}
  [119] = {x=92.587528, y=38.348029, z=37.091522, rx=-0.277717, ry=-89.960922, rz=89.722393, shoulder=lefty, elbow=epositive, wrist=wpositive, fatherId=frmaster[1]}
  [120] = {x=93.786865, y=38.763402, z=33.795174, rx=0.006902, ry=-87.932967, rz=90.007139, shoulder=lefty, elbow=epositive, wrist=wpositive, fatherId=frmaster[1]}
  [121] = {x=94.683389, y=39.18394, z=31.030856, rx=-0.007201, ry=-86.250705, rz=89.992934, shoulder=lefty, elbow=epositive, wrist=wpositive, fatherId=frmaster[1]}
  [122] = {x=95.333429, y=39.599226, z=28.809223, rx=-0.000946, ry=-84.914855, rz=89.999411, shoulder=lefty, elbow=epositive, wrist=wpositive, fatherId=frmaster[1]}
  [123] = {x=96.08972, y=41.269963, z=25.405902, rx=-0.004395, ry=-82.881448, rz=89.9952, shoulder=lefty, elbow=epositive, wrist=wpositive, fatherId=frmaster[1]}
  [124] = {x=95.935268, y=42.915477, z=24.779711, rx=0.000881, ry=-82.503167, rz=90.000833, shoulder=lefty, elbow=epositive, wrist=wpositive, fatherId=frmaster[1]}
  [125] = {x=96.100323, y=44.566138, z=22.828786, rx=-0.002191, ry=-81.339159, rz=89.998314, shoulder=lefty, elbow=epositive, wrist=wpositive, fatherId=frmaster[1]}
  [126] = {x=96.256227, y=46.202919, z=20.293043, rx=-0.001708, ry=-79.828293, rz=89.99802, shoulder=lefty, elbow=epositive, wrist=wpositive, fatherId=frmaster[1]}
  [127] = {x=95.997279, y=47.836326, z=19.528446, rx=-0.002303, ry=-79.373746, rz=89.998285, shoulder=lefty, elbow=epositive, wrist=wpositive, fatherId=frmaster[1]}
  [128] = {x=95.511093, y=49.449252, z=19.530551, rx=-0.001558, ry=-79.373174, rz=89.998921, shoulder=lefty, elbow=epositive, wrist=wpositive, fatherId=frmaster[1]}
  [129] = {x=95.027362, y=51.065454, z=19.527338, rx=0.000846, ry=-79.374158, rz=90.00015, shoulder=lefty, elbow=epositive, wrist=wpositive, fatherId=frmaster[1]}
  [130] = {x=94.482438, y=52.662308, z=19.532609, rx=-0.004337, ry=-79.37314, rz=89.996111, shoulder=lefty, elbow=epositive, wrist=wpositive, fatherId=frmaster[1]}
  [131] = {x=93.944444, y=54.256316, z=19.52564, rx=0.003031, ry=-79.374288, rz=90.002788, shoulder=lefty, elbow=epositive, wrist=wpositive, fatherId=frmaster[1]}
  [132] = {x=93.358928, y=55.841946, z=19.530243, rx=-0.003919, ry=-79.373341, rz=89.996606, shoulder=lefty, elbow=epositive, wrist=wpositive, fatherId=frmaster[1]}
  [133] = {x=92.778971, y=57.424452, z=19.529688, rx=0.001054, ry=-79.373683, rz=90.000971, shoulder=lefty, elbow=epositive, wrist=wpositive, fatherId=frmaster[1]}
  [134] = {x=91.958358, y=59.52389, z=19.527648, rx=0.000464, ry=-79.374052, rz=90.00036, shoulder=lefty, elbow=epositive, wrist=wpositive, fatherId=frmaster[1]}
  [135] = {x=91.141615, y=61.619681, z=19.527131, rx=-0.000671, ry=-79.373951, rz=89.999459, shoulder=lefty, elbow=epositive, wrist=wpositive, fatherId=frmaster[1]}
  [136] = {x=90.325218, y=63.715632, z=19.527445, rx=0.003861, ry=-79.373934, rz=90.003796, shoulder=lefty, elbow=epositive, wrist=wpositive, fatherId=frmaster[1]}
  [137] = {x=91.094649, y=61.564128, z=19.526589, rx=0.003855, ry=-79.373896, rz=90.003237, shoulder=lefty, elbow=epositive, wrist=wpositive, fatherId=frmaster[1]}
  [138] = {x=91.861106, y=59.410958, z=19.529598, rx=0.003973, ry=-79.373359, rz=90.004251, shoulder=lefty, elbow=epositive, wrist=wpositive, fatherId=frmaster[1]}
  [139] = {x=92.573792, y=57.240499, z=19.532382, rx=0.003356, ry=-79.372933, rz=90.003953, shoulder=lefty, elbow=epositive, wrist=wpositive, fatherId=frmaster[1]}
  [140] = {x=93.289164, y=55.070447, z=19.528713, rx=0.00408, ry=-79.373804, rz=90.004578, shoulder=lefty, elbow=epositive, wrist=wpositive, fatherId=frmaster[1]}
  [141] = {x=93.951014, y=52.889778, z=19.529948, rx=-0.002079, ry=-79.373903, rz=89.997873, shoulder=lefty, elbow=epositive, wrist=wpositive, fatherId=frmaster[1]}
  [142] = {x=94.611871, y=50.705065, z=19.528364, rx=-0.002, ry=-79.374279, rz=89.998338, shoulder=lefty, elbow=epositive, wrist=wpositive, fatherId=frmaster[1]}
  [143] = {x=95.220498, y=48.499121, z=19.528287, rx=0.00203, ry=-79.373757, rz=90.002331, shoulder=lefty, elbow=epositive, wrist=wpositive, fatherId=frmaster[1]}
  [144] = {x=95.827788, y=46.297382, z=19.529092, rx=0.001975, ry=-79.373784, rz=90.00247, shoulder=lefty, elbow=epositive, wrist=wpositive, fatherId=frmaster[1]}
  [145] = {x=96.263857, y=44.083642, z=20.098112, rx=-0.004052, ry=-79.713472, rz=89.995488, shoulder=lefty, elbow=epositive, wrist=wpositive, fatherId=frmaster[1]}
  [146] = {x=96.050371, y=41.86495, z=23.490709, rx=0.002624, ry=-81.734706, rz=90.002672, shoulder=lefty, elbow=epositive, wrist=wpositive, fatherId=frmaster[1]}
  [147] = {x=96.037873, y=39.642192, z=25.529927, rx=-0.002642, ry=-82.954597, rz=89.997083, shoulder=lefty, elbow=epositive, wrist=wpositive, fatherId=frmaster[1]}
  [148] = {x=95.186271, y=38.522912, z=29.329009, rx=0.002173, ry=-85.224913, rz=90.002691, shoulder=lefty, elbow=epositive, wrist=wpositive, fatherId=frmaster[1]}
  [149] = {x=94.346619, y=38.244969, z=32.111867, rx=-0.007895, ry=-86.910603, rz=89.992176, shoulder=lefty, elbow=epositive, wrist=wpositive, fatherId=frmaster[1]}
  [150] = {x=93.127959, y=37.962188, z=35.653832, rx=0.044273, ry=-89.071005, rz=90.044474, shoulder=lefty, elbow=epositive, wrist=wpositive, fatherId=frmaster[1]}
  [151] = {x=91.447601, y=37.683514, z=39.906836, rx=-0.001307, ry=-91.709649, rz=89.998762, shoulder=lefty, elbow=epositive, wrist=wpositive, fatherId=frmaster[1]}
  [152] = {x=90.407577, y=37.550026, z=42.270107, rx=-179.991776, ry=-86.795951, rz=-89.992541, shoulder=lefty, elbow=epositive, wrist=wpositive, fatherId=frmaster[1]}
  [153] = {x=89.222759, y=37.407078, z=44.7793, rx=-0.004467, ry=-94.80646, rz=89.994509, shoulder=lefty, elbow=epositive, wrist=wpositive, fatherId=frmaster[1]}
  [154] = {x=87.122839, y=37.130069, z=48.841923, rx=-179.996935, ry=-82.555967, rz=-89.9968, shoulder=lefty, elbow=epositive, wrist=wpositive, fatherId=frmaster[1]}
  [155] = {x=85.096513, y=36.850159, z=52.391129, rx=-0.000158, ry=-99.803001, rz=89.999789, shoulder=lefty, elbow=epositive, wrist=wpositive, fatherId=frmaster[1]}
  [156] = {x=82.997863, y=36.568675, z=55.745289, rx=-0.001539, ry=-102.092476, rz=89.997873, shoulder=lefty, elbow=epositive, wrist=wpositive, fatherId=frmaster[1]}
  [157] = {x=80.846236, y=36.28753, z=58.904638, rx=-0.003263, ry=-104.297303, rz=89.996904, shoulder=lefty, elbow=epositive, wrist=wpositive, fatherId=frmaster[1]}
  [158] = {x=78.679239, y=36.013365, z=61.84087, rx=-0.000009, ry=-106.410297, rz=89.999912, shoulder=lefty, elbow=epositive, wrist=wpositive, fatherId=frmaster[1]}
  [159] = {x=76.513869, y=35.734897, z=64.569571, rx=0.000474, ry=-108.423914, rz=89.999877, shoulder=lefty, elbow=epositive, wrist=wpositive, fatherId=frmaster[1]}
  [160] = {x=74.377516, y=35.455256, z=67.084647, rx=0.00029, ry=-110.337342, rz=89.99988, shoulder=lefty, elbow=epositive, wrist=wpositive, fatherId=frmaster[1]}
  [161] = {x=72.272486, y=35.176813, z=69.410781, rx=-179.999659, ry=-67.852996, rz=-89.999407, shoulder=lefty, elbow=epositive, wrist=wpositive, fatherId=frmaster[1]}
  [162] = {x=70.114435, y=34.895064, z=71.650249, rx=-0.000221, ry=-113.953974, rz=89.999587, shoulder=lefty, elbow=epositive, wrist=wpositive, fatherId=frmaster[1]}
  [163] = {x=67.983278, y=34.614496, z=73.730252, rx=-0.001701, ry=-115.680892, rz=89.997951, shoulder=lefty, elbow=epositive, wrist=wpositive, fatherId=frmaster[1]}
  [164] = {x=65.897706, y=34.33711, z=75.654004, rx=-0.000849, ry=-117.327184, rz=89.99874, shoulder=lefty, elbow=epositive, wrist=wpositive, fatherId=frmaster[1]}
  [165] = {x=63.860879, y=34.058625, z=77.430804, rx=-0.001116, ry=-118.893435, rz=89.998692, shoulder=lefty, elbow=epositive, wrist=wpositive, fatherId=frmaster[1]}
  [166] = {x=59.980715, y=33.506732, z=80.567486, rx=-179.998605, ry=-58.205492, rz=-89.998427, shoulder=lefty, elbow=epositive, wrist=wpositive, fatherId=frmaster[1]}
  [167] = {x=56.366769, y=32.945365, z=83.222104, rx=179.99942, ry=-55.592706, rz=-89.999616, shoulder=lefty, elbow=epositive, wrist=wpositive, fatherId=frmaster[1]}
  [168] = {x=52.823453, y=32.389192, z=85.594722, rx=179.99947, ry=-53.10386, rz=-89.99992, shoulder=lefty, elbow=epositive, wrist=wpositive, fatherId=frmaster[1]}
  [169] = {x=49.5295, y=31.831729, z=87.61192, rx=-0.000223, ry=-129.161992, rz=89.999857, shoulder=lefty, elbow=epositive, wrist=wpositive, fatherId=frmaster[1]}
  [170] = {x=46.464539, y=31.280612, z=89.343462, rx=-179.99971, ry=-48.774585, rz=-89.999859, shoulder=lefty, elbow=epositive, wrist=wpositive, fatherId=frmaster[1]}
  [171] = {x=43.623245, y=30.722081, z=90.825772, rx=-179.999587, ry=-46.887235, rz=-89.999769, shoulder=lefty, elbow=epositive, wrist=wpositive, fatherId=frmaster[1]}
  [172] = {x=40.816813, y=30.169325, z=92.181981, rx=-179.99942, ry=-45.047713, rz=-89.99954, shoulder=lefty, elbow=epositive, wrist=wpositive, fatherId=frmaster[1]}
  [173] = {x=38.35747, y=29.612371, z=93.286769, rx=0.000088, ry=-136.554977, rz=89.999788, shoulder=lefty, elbow=epositive, wrist=wpositive, fatherId=frmaster[1]}
  [174] = {x=34.151211, y=28.505863, z=95.006361, rx=0.000392, ry=-139.275461, rz=89.999831, shoulder=lefty, elbow=epositive, wrist=wpositive, fatherId=frmaster[1]}
  [175] = {x=29.583315, y=27.395817, z=96.625929, rx=179.999636, ry=-37.826372, rz=-89.999897, shoulder=lefty, elbow=epositive, wrist=wpositive, fatherId=frmaster[1]}
  [176] = {x=24.846184, y=26.288373, z=98.026387, rx=-0.000386, ry=-145.126226, rz=89.999677, shoulder=lefty, elbow=epositive, wrist=wpositive, fatherId=frmaster[1]}
  [177] = {x=22.318326, y=25.738171, z=98.668559, rx=-0.00035, ry=-146.685517, rz=89.999636, shoulder=lefty, elbow=epositive, wrist=wpositive, fatherId=frmaster[1]}
  [178] = {x=19.725634, y=25.190914, z=99.254652, rx=-179.999814, ry=-31.731612, rz=-89.998701, shoulder=lefty, elbow=epositive, wrist=wpositive, fatherId=frmaster[1]}
  [179] = {x=17.065248, y=24.640618, z=99.764539, rx=-179.998876, ry=-30.113055, rz=-89.999198, shoulder=lefty, elbow=epositive, wrist=wpositive, fatherId=frmaster[1]}
  [180] = {x=14.339161, y=24.083611, z=100.219022, rx=0.000391, ry=-151.532808, rz=89.999546, shoulder=lefty, elbow=epositive, wrist=wpositive, fatherId=frmaster[1]}
  [181] = {x=11.265133, y=23.535787, z=100.634249, rx=-0.000566, ry=-153.375984, rz=89.999231, shoulder=lefty, elbow=epositive, wrist=wpositive, fatherId=frmaster[1]}
  [182] = {x=6.689955, y=22.99633, z=101.051081, rx=-179.999802, ry=-23.932717, rz=-89.999477, shoulder=lefty, elbow=epositive, wrist=wpositive, fatherId=frmaster[1]}
  [183] = {x=2.558295, y=22.594575, z=101.247419, rx=0.000587, ry=-158.489238, rz=89.999927, shoulder=lefty, elbow=epositive, wrist=wpositive, fatherId=frmaster[1]}
  [184] = {x=-1.276075, y=22.192451, z=101.275185, rx=179.999672, ry=-19.261277, rz=-89.9999, shoulder=lefty, elbow=epositive, wrist=wpositive, fatherId=frmaster[1]}
  [185] = {x=-5.510672, y=21.810678, z=101.124148, rx=-179.999971, ry=-16.766605, rz=-89.999255, shoulder=lefty, elbow=epositive, wrist=wpositive, fatherId=frmaster[1]}
  [186] = {x=-9.301027, y=21.420367, z=100.842326, rx=-0.000846, ry=-165.479966, rz=89.99971, shoulder=lefty, elbow=epositive, wrist=wpositive, fatherId=frmaster[1]}
  [187] = {x=-13.456621, y=21.062192, z=100.345172, rx=-179.999947, ry=-12.030124, rz=-89.999229, shoulder=lefty, elbow=epositive, wrist=wpositive, fatherId=frmaster[1]}
  [188] = {x=-16.96517, y=20.696133, z=99.775069, rx=0.000401, ry=-170.105369, rz=89.999567, shoulder=lefty, elbow=epositive, wrist=wpositive, fatherId=frmaster[1]}
  [189] = {x=-20.671992, y=20.383174, z=99.021029, rx=-0.00001, ry=-172.407267, rz=89.999814, shoulder=lefty, elbow=epositive, wrist=wpositive, fatherId=frmaster[1]}
  [190] = {x=-23.232028, y=20.080629, z=98.387818, rx=0.00043, ry=-174.056533, rz=89.999908, shoulder=lefty, elbow=epositive, wrist=wpositive, fatherId=frmaster[1]}
  [191] = {x=-23.232149, y=20.079538, z=108.391214, rx=179.999501, ry=-5.943638, rz=-89.999813, shoulder=lefty, elbow=epositive, wrist=wpositive, fatherId=frmaster[1]}
  [192] = {x=-18.610941, y=20.073872, z=152.751749, rx=-0.000319, ry=-174.055977, rz=89.999195, shoulder=lefty, elbow=epositive, wrist=wpositive, fatherId=frmaster[1]}
  [193] = {x=-58.457155, y=-2.837264, z=156.675838, rx=0.000195, ry=-174.221721, rz=-0.000461, shoulder=lefty, elbow=epositive, wrist=wpositive, fatherId=frmaster[1]}
  [194] = {x=-62.950739, y=-2.831421, z=112.320225, rx=-0.000098, ry=-174.220553, rz=0.000511, shoulder=lefty, elbow=epositive, wrist=wpositive, fatherId=frmaster[1]}
  [195] = {x=-62.948805, y=-2.831104, z=102.322171, rx=-0.000194, ry=-174.221362, rz=0.000974, shoulder=lefty, elbow=epositive, wrist=wpositive, fatherId=frmaster[1]}
  [196] = {x=-59.331081, y=-2.911163, z=104.643589, rx=0.000307, ry=-172.04671, rz=0.000002, shoulder=lefty, elbow=epositive, wrist=wpositive, fatherId=frmaster[1]}
  [197] = {x=-54.81737, y=-2.994006, z=107.245031, rx=-0.000408, ry=-169.436929, rz=0.000571, shoulder=lefty, elbow=epositive, wrist=wpositive, fatherId=frmaster[1]}
  [198] = {x=-51.807758, y=-3.044147, z=108.77684, rx=-0.00002, ry=-167.785225, rz=0.000385, shoulder=lefty, elbow=epositive, wrist=wpositive, fatherId=frmaster[1]}
  [199] = {x=-48.780926, y=-3.091436, z=110.224119, rx=-0.00047, ry=-166.143283, rz=0.000496, shoulder=lefty, elbow=epositive, wrist=wpositive, fatherId=frmaster[1]}
  [200] = {x=-45.730052, y=-3.141145, z=111.570995, rx=-0.000239, ry=-164.510841, rz=0.000407, shoulder=lefty, elbow=epositive, wrist=wpositive, fatherId=frmaster[1]}
  [201] = {x=-42.65424, y=-3.192333, z=112.812629, rx=0.000556, ry=-162.887217, rz=-0.000805, shoulder=lefty, elbow=epositive, wrist=wpositive, fatherId=frmaster[1]}
  [202] = {x=-39.754901, y=-3.256157, z=113.911808, rx=-0.000549, ry=-161.367851, rz=-0.000341, shoulder=lefty, elbow=epositive, wrist=wpositive, fatherId=frmaster[1]}
  [203] = {x=-36.817365, y=-3.310227, z=114.923732, rx=0.000425, ry=-159.846521, rz=0.000113, shoulder=lefty, elbow=epositive, wrist=wpositive, fatherId=frmaster[1]}
  [204] = {x=-33.840125, y=-3.373804, z=115.87198, rx=0.000416, ry=-158.31717, rz=-0.000003, shoulder=lefty, elbow=epositive, wrist=wpositive, fatherId=frmaster[1]}
  [205] = {x=-30.823918, y=-3.436002, z=116.733606, rx=0.000569, ry=-156.781875, rz=0.00044, shoulder=lefty, elbow=epositive, wrist=wpositive, fatherId=frmaster[1]}
  [206] = {x=-25.459936, y=-3.596747, z=118.065788, rx=-0.000203, ry=-154.078894, rz=-0.000535, shoulder=lefty, elbow=epositive, wrist=wpositive, fatherId=frmaster[1]}
  [207] = {x=-19.888542, y=-3.755603, z=119.163649, rx=-0.000413, ry=-151.3029, rz=-0.000683, shoulder=lefty, elbow=epositive, wrist=wpositive, fatherId=frmaster[1]}
  [208] = {x=-14.103877, y=-3.906494, z=120.012057, rx=0.000607, ry=-148.446877, rz=0.000414, shoulder=lefty, elbow=epositive, wrist=wpositive, fatherId=frmaster[1]}
  [209] = {x=-8.109169, y=-4.064105, z=120.575929, rx=0.000148, ry=-145.508211, rz=-0.000427, shoulder=lefty, elbow=epositive, wrist=wpositive, fatherId=frmaster[1]}
  [210] = {x=-2.35706, y=-4.158909, z=120.828178, rx=0.000209, ry=-142.744473, rz=-0.000933, shoulder=lefty, elbow=epositive, wrist=wpositive, fatherId=frmaster[1]}
  [211] = {x=0.814019, y=-4.187101, z=120.855975, rx=0.000045, ry=-141.226564, rz=0.000207, shoulder=lefty, elbow=epositive, wrist=wpositive, fatherId=frmaster[1]}
  [212] = {x=6.815598, y=-4.251946, z=120.665364, rx=-0.000072, ry=-138.357327, rz=-0.000552, shoulder=lefty, elbow=epositive, wrist=wpositive, fatherId=frmaster[1]}
  [213] = {x=12.263488, y=-4.309628, z=120.226681, rx=0.000825, ry=-135.743522, rz=0.000868, shoulder=lefty, elbow=epositive, wrist=wpositive, fatherId=frmaster[1]}
  [214] = {x=17.104551, y=-4.374383, z=119.631034, rx=0.00019, ry=-133.407549, rz=-0.000143, shoulder=lefty, elbow=epositive, wrist=wpositive, fatherId=frmaster[1]}
  [215] = {x=21.319008, y=-4.437937, z=118.94273, rx=-0.000709, ry=-131.359302, rz=0.000004, shoulder=lefty, elbow=epositive, wrist=wpositive, fatherId=frmaster[1]}
  [216] = {x=24.91966, y=-4.499109, z=118.231178, rx=-0.000464, ry=-129.594656, rz=-0.000196, shoulder=lefty, elbow=epositive, wrist=wpositive, fatherId=frmaster[1]}
  [217] = {x=27.937112, y=-4.558493, z=117.545843, rx=0.001022, ry=-128.104076, rz=0.000525, shoulder=lefty, elbow=epositive, wrist=wpositive, fatherId=frmaster[1]}
  [218] = {x=33.536787, y=-4.756391, z=116.033047, rx=-0.000023, ry=-125.292591, rz=-0.000126, shoulder=lefty, elbow=epositive, wrist=wpositive, fatherId=frmaster[1]}
  [219] = {x=38.733004, y=-5.348967, z=114.284126, rx=-0.000501, ry=-122.507552, rz=-0.000666, shoulder=lefty, elbow=epositive, wrist=wpositive, fatherId=frmaster[1]}
  [220] = {x=42.913654, y=-5.449118, z=112.758097, rx=-0.000522, ry=-120.366833, rz=-0.000447, shoulder=lefty, elbow=epositive, wrist=wpositive, fatherId=frmaster[1]}
  [221] = {x=46.958105, y=-5.553398, z=111.106726, rx=-0.000259, ry=-118.263864, rz=0.000087, shoulder=lefty, elbow=epositive, wrist=wpositive, fatherId=frmaster[1]}
  [222] = {x=50.870719, y=-5.657003, z=109.346844, rx=-0.000938, ry=-116.199505, rz=-0.000413, shoulder=lefty, elbow=epositive, wrist=wpositive, fatherId=frmaster[1]}
  [223] = {x=54.640258, y=-5.753393, z=107.479195, rx=0.001053, ry=-114.173024, rz=0.000403, shoulder=lefty, elbow=epositive, wrist=wpositive, fatherId=frmaster[1]}
  [224] = {x=58.28046, y=-5.858883, z=105.518617, rx=-0.000073, ry=-112.182529, rz=0.000285, shoulder=lefty, elbow=epositive, wrist=wpositive, fatherId=frmaster[1]}
  [225] = {x=61.78664, y=-5.961639, z=103.465034, rx=-0.000994, ry=-110.225888, rz=-0.000641, shoulder=lefty, elbow=epositive, wrist=wpositive, fatherId=frmaster[1]}
  [226] = {x=65.166577, y=-6.059206, z=101.331147, rx=-0.000055, ry=-108.298622, rz=0.000138, shoulder=lefty, elbow=epositive, wrist=wpositive, fatherId=frmaster[1]}
  [227] = {x=68.431563, y=-6.166454, z=99.114483, rx=-0.001184, ry=-106.397685, rz=-0.000473, shoulder=lefty, elbow=epositive, wrist=wpositive, fatherId=frmaster[1]}
  [228] = {x=72.501095, y=-6.302935, z=96.122058, rx=-0.001612, ry=-103.962248, rz=-0.0017, shoulder=lefty, elbow=epositive, wrist=wpositive, fatherId=frmaster[1]}
  [229] = {x=76.463906, y=-6.434972, z=92.929435, rx=0.002158, ry=-101.512143, rz=0.0013, shoulder=lefty, elbow=epositive, wrist=wpositive, fatherId=frmaster[1]}
  [230] = {x=79.670568, y=-6.577069, z=90.12947, rx=-0.003997, ry=-99.455729, rz=-0.004414, shoulder=lefty, elbow=epositive, wrist=wpositive, fatherId=frmaster[1]}
  [231] = {x=81.195641, y=-6.71291, z=88.684389, rx=-0.001718, ry=-98.426232, rz=-0.002303, shoulder=lefty, elbow=epositive, wrist=wpositive, fatherId=frmaster[1]}
  [232] = {x=84.061723, y=-6.986336, z=85.817261, rx=0.002607, ry=-96.439473, rz=0.00219, shoulder=lefty, elbow=epositive, wrist=wpositive, fatherId=frmaster[1]}
  [233] = {x=86.682122, y=-7.259848, z=83.011655, rx=0.007979, ry=-94.550869, rz=0.008977, shoulder=lefty, elbow=epositive, wrist=wpositive, fatherId=frmaster[1]}
  [234] = {x=89.095474, y=-7.537365, z=80.239467, rx=0.000927, ry=-92.745892, rz=0.000718, shoulder=lefty, elbow=epositive, wrist=wpositive, fatherId=frmaster[1]}
  [235] = {x=91.308993, y=-7.811203, z=77.521772, rx=-0.029514, ry=-91.025881, rz=-0.030692, shoulder=lefty, elbow=epositive, wrist=wpositive, fatherId=frmaster[1]}
  [236] = {x=93.32424, y=-8.085724, z=74.889294, rx=-0.008484, ry=-89.388383, rz=-0.009305, shoulder=lefty, elbow=epositive, wrist=wpositive, fatherId=frmaster[1]}
  [237] = {x=95.160856, y=-8.363212, z=72.340007, rx=0.014263, ry=-87.836718, rz=0.014604, shoulder=lefty, elbow=epositive, wrist=wpositive, fatherId=frmaster[1]}
  [238] = {x=98.432797, y=-8.91116, z=67.348232, rx=0.000761, ry=-84.884513, rz=0.000669, shoulder=lefty, elbow=epositive, wrist=wpositive, fatherId=frmaster[1]}
  [239] = {x=101.122184, y=-9.453559, z=62.710795, rx=-0.001427, ry=-82.22321, rz=-0.001903, shoulder=lefty, elbow=epositive, wrist=wpositive, fatherId=frmaster[1]}
  [240] = {x=103.312693, y=-10.00312, z=58.459619, rx=0.000333, ry=-79.835437, rz=0.000889, shoulder=lefty, elbow=epositive, wrist=wpositive, fatherId=frmaster[1]}
  [241] = {x=105.090295, y=-10.552695, z=54.578282, rx=0.001131, ry=-77.703403, rz=0.001569, shoulder=lefty, elbow=epositive, wrist=wpositive, fatherId=frmaster[1]}
  [242] = {x=103.840447, y=-12.708609, z=54.354496, rx=-0.003676, ry=-77.581665, rz=-0.003378, shoulder=lefty, elbow=epositive, wrist=wpositive, fatherId=frmaster[1]}
  [243] = {x=102.445667, y=-14.852462, z=54.348712, rx=0.000104, ry=-77.582565, rz=0.000154, shoulder=lefty, elbow=epositive, wrist=wpositive, fatherId=frmaster[1]}
  [244] = {x=101.01074, y=-16.970168, z=54.353831, rx=-0.002926, ry=-77.582005, rz=-0.002307, shoulder=lefty, elbow=epositive, wrist=wpositive, fatherId=frmaster[1]}
  [245] = {x=99.548937, y=-19.06947, z=54.350705, rx=-0.001699, ry=-77.582192, rz=-0.001475, shoulder=lefty, elbow=epositive, wrist=wpositive, fatherId=frmaster[1]}
  [246] = {x=98.057167, y=-21.141825, z=54.350832, rx=-0.001367, ry=-77.582283, rz=-0.002023, shoulder=lefty, elbow=epositive, wrist=wpositive, fatherId=frmaster[1]}
  [247] = {x=96.534028, y=-23.197602, z=54.354616, rx=0.00199, ry=-77.581438, rz=0.001672, shoulder=lefty, elbow=epositive, wrist=wpositive, fatherId=frmaster[1]}
  [248] = {x=97.641783, y=-22.006556, z=54.357129, rx=-0.001972, ry=-77.581234, rz=-0.001753, shoulder=lefty, elbow=epositive, wrist=wpositive, fatherId=frmaster[1]}
  [249] = {x=98.754973, y=-20.813399, z=54.353693, rx=-0.002893, ry=-77.581817, rz=-0.002603, shoulder=lefty, elbow=epositive, wrist=wpositive, fatherId=frmaster[1]}
  [250] = {x=99.862379, y=-19.61902, z=54.351705, rx=-0.000678, ry=-77.582227, rz=-0.000971, shoulder=lefty, elbow=epositive, wrist=wpositive, fatherId=frmaster[1]}
  [251] = {x=100.971416, y=-18.425872, z=54.355533, rx=0.003257, ry=-77.581919, rz=0.003227, shoulder=lefty, elbow=epositive, wrist=wpositive, fatherId=frmaster[1]}
  [252] = {x=102.048613, y=-17.206038, z=54.35678, rx=-0.00229, ry=-77.58165, rz=-0.001959, shoulder=lefty, elbow=epositive, wrist=wpositive, fatherId=frmaster[1]}
  [253] = {x=103.128246, y=-15.988358, z=54.356549, rx=-0.00129, ry=-77.581082, rz=-0.00072, shoulder=lefty, elbow=epositive, wrist=wpositive, fatherId=frmaster[1]}
  [254] = {x=104.137439, y=-14.718625, z=54.350754, rx=0.001734, ry=-77.582513, rz=0.001665, shoulder=lefty, elbow=epositive, wrist=wpositive, fatherId=frmaster[1]}
  [255] = {x=105.055392, y=-13.37907, z=54.354263, rx=-0.003561, ry=-77.581593, rz=-0.003116, shoulder=lefty, elbow=epositive, wrist=wpositive, fatherId=frmaster[1]}
  [256] = {x=103.82803, y=-12.682327, z=57.373699, rx=0.001185, ry=-79.240345, rz=0.000884, shoulder=lefty, elbow=epositive, wrist=wpositive, fatherId=frmaster[1]}
  [257] = {x=101.330649, y=-11.986221, z=62.329516, rx=-0.001375, ry=-82.002258, rz=-0.001362, shoulder=lefty, elbow=epositive, wrist=wpositive, fatherId=frmaster[1]}
  [258] = {x=98.923844, y=-11.249065, z=66.539032, rx=0.005094, ry=-84.41488, rz=0.004688, shoulder=lefty, elbow=epositive, wrist=wpositive, fatherId=frmaster[1]}
  [259] = {x=96.915412, y=-10.487034, z=69.741857, rx=0.003624, ry=-86.283948, rz=0.004634, shoulder=lefty, elbow=epositive, wrist=wpositive, fatherId=frmaster[1]}
  [260] = {x=95.920101, y=-9.135764, z=71.233256, rx=-0.003973, ry=-87.173203, rz=-0.003996, shoulder=lefty, elbow=epositive, wrist=wpositive, fatherId=frmaster[1]}
  [261] = {x=98.341691, y=-8.06863, z=67.489874, rx=-0.003359, ry=-84.96843, rz=-0.004037, shoulder=lefty, elbow=epositive, wrist=wpositive, fatherId=frmaster[1]}
  [262] = {x=100.773293, y=-7.488613, z=63.349887, rx=0.000768, ry=-82.583389, rz=0.001539, shoulder=lefty, elbow=epositive, wrist=wpositive, fatherId=frmaster[1]}
  [263] = {x=102.399, y=-7.164342, z=60.297929, rx=0.00074, ry=-80.862239, rz=0.000551, shoulder=lefty, elbow=epositive, wrist=wpositive, fatherId=frmaster[1]}
  [264] = {x=103.805852, y=-6.837764, z=57.431094, rx=0.001667, ry=-79.269638, rz=0.002006, shoulder=lefty, elbow=epositive, wrist=wpositive, fatherId=frmaster[1]}
  [265] = {x=104.908102, y=-6.259088, z=54.352077, rx=0.001069, ry=-77.58207, rz=0.001031, shoulder=lefty, elbow=epositive, wrist=wpositive, fatherId=frmaster[1]}
  [266] = {x=103.026172, y=-4.762106, z=54.348312, rx=0.00024, ry=-77.582304, rz=-0.000748, shoulder=lefty, elbow=epositive, wrist=wpositive, fatherId=frmaster[1]}
  [267] = {x=100.981976, y=-3.483489, z=54.350188, rx=0.002978, ry=-77.582284, rz=0.002626, shoulder=lefty, elbow=epositive, wrist=wpositive, fatherId=frmaster[1]}
  [268] = {x=99.594968, y=-2.651669, z=54.355787, ry=-77.581361, rz=0.000498, shoulder=lefty, elbow=epositive, wrist=wpositive, fatherId=frmaster[1]}
  [269] = {x=98.23614, y=-1.766761, z=54.351028, rx=-0.00175, ry=-77.581702, rz=-0.001543, shoulder=lefty, elbow=epositive, wrist=wpositive, fatherId=frmaster[1]}
  [270] = {x=97.124249, y=-0.903418, z=54.351052, rx=0.000806, ry=-77.581911, rz=0.001115, shoulder=lefty, elbow=epositive, wrist=wpositive, fatherId=frmaster[1]}
  [271] = {x=96.537342, y=-0.232614, z=54.35059, rx=-0.000215, ry=-77.582299, rz=-0.000088, shoulder=lefty, elbow=epositive, wrist=wpositive, fatherId=frmaster[1]}
  [272] = {x=96.311447, y=0.155702, z=54.356044, rx=-0.001724, ry=-77.581159, rz=-0.001306, shoulder=lefty, elbow=epositive, wrist=wpositive, fatherId=frmaster[1]}
  [273] = {x=96.172638, y=0.965831, z=54.348171, rx=-0.003705, ry=-77.582722, rz=-0.003982, shoulder=lefty, elbow=epositive, wrist=wpositive, fatherId=frmaster[1]}
  [274] = {x=96.378457, y=1.662687, z=54.352798, rx=-0.000893, ry=-77.582071, rz=-0.000654, shoulder=lefty, elbow=epositive, wrist=wpositive, fatherId=frmaster[1]}
  [275] = {x=96.716004, y=2.209968, z=54.358295, rx=-0.001932, ry=-77.580912, rz=-0.001546, shoulder=lefty, elbow=epositive, wrist=wpositive, fatherId=frmaster[1]}
  [276] = {x=97.145819, y=2.701623, z=54.350675, rx=0.002898, ry=-77.582304, rz=0.003113, shoulder=lefty, elbow=epositive, wrist=wpositive, fatherId=frmaster[1]}
  [277] = {x=98.135394, y=3.570119, z=54.351347, rx=0.001312, ry=-77.582356, rz=0.001769, shoulder=lefty, elbow=epositive, wrist=wpositive, fatherId=frmaster[1]}
  [278] = {x=100.271915, y=5.145232, z=54.354772, rx=0.000774, ry=-77.581495, rz=0.001138, shoulder=lefty, elbow=epositive, wrist=wpositive, fatherId=frmaster[1]}
  [279] = {x=101.613209, y=6.055404, z=54.355209, rx=-0.001767, ry=-77.581775, rz=-0.001154, shoulder=lefty, elbow=epositive, wrist=wpositive, fatherId=frmaster[1]}
  [280] = {x=102.954606, y=6.966263, z=54.354139, rx=-0.002387, ry=-77.58191, rz=-0.00257, shoulder=lefty, elbow=epositive, wrist=wpositive, fatherId=frmaster[1]}
  [281] = {x=104.257281, y=7.92866, z=54.34828, rx=0.001512, ry=-77.582295, rz=0.00145, shoulder=lefty, elbow=epositive, wrist=wpositive, fatherId=frmaster[1]}
  [282] = {x=103.648294, y=8.99161, z=57.758028, rx=-0.00367, ry=-79.450811, rz=-0.004045, shoulder=lefty, elbow=epositive, wrist=wpositive, fatherId=frmaster[1]}
  [283] = {x=101.924592, y=9.281593, z=61.214887, rx=-0.001172, ry=-81.374361, rz=-0.001232, shoulder=lefty, elbow=epositive, wrist=wpositive, fatherId=frmaster[1]}
  [284] = {x=99.878062, y=9.577681, z=64.92308, rx=-0.007231, ry=-83.484301, rz=-0.007603, shoulder=lefty, elbow=epositive, wrist=wpositive, fatherId=frmaster[1]}
  [285] = {x=98.08671, y=9.853504, z=67.905684, rx=-0.006037, ry=-85.206465, rz=-0.006041, shoulder=lefty, elbow=epositive, wrist=wpositive, fatherId=frmaster[1]}
  [286] = {x=96.058356, y=10.1293, z=71.027182, rx=-0.000074, ry=-87.050089, rz=0.000133, shoulder=lefty, elbow=epositive, wrist=wpositive, fatherId=frmaster[1]}
  [287] = {x=94.234705, y=10.429232, z=73.648524, rx=0.011775, ry=-88.628725, rz=0.012476, shoulder=lefty, elbow=epositive, wrist=wpositive, fatherId=frmaster[1]}
  [288] = {x=92.222876, y=10.73188, z=76.35399, rx=-0.030619, ry=-90.292386, rz=-0.030725, shoulder=lefty, elbow=epositive, wrist=wpositive, fatherId=frmaster[1]}
  [289] = {x=89.818157, y=11.221312, z=79.372538, rx=-0.017833, ry=-92.195305, rz=-0.018494, shoulder=lefty, elbow=epositive, wrist=wpositive, fatherId=frmaster[1]}
  [290] = {x=87.882125, y=12.107701, z=81.657728, rx=-0.001083, ry=-93.663451, rz=-0.000711, shoulder=lefty, elbow=epositive, wrist=wpositive, fatherId=frmaster[1]}
  [291] = {x=89.988148, y=13.286016, z=79.167902, rx=-0.004645, ry=-92.062035, rz=-0.004366, shoulder=lefty, elbow=epositive, wrist=wpositive, fatherId=frmaster[1]}
  [292] = {x=93.367569, y=14.021359, z=74.829658, rx=0.022945, ry=-89.354004, rz=0.022742, shoulder=lefty, elbow=epositive, wrist=wpositive, fatherId=frmaster[1]}
  [293] = {x=95.402493, y=14.365041, z=71.990028, rx=0.01328, ry=-87.625641, rz=0.013771, shoulder=lefty, elbow=epositive, wrist=wpositive, fatherId=frmaster[1]}
  [294] = {x=97.234085, y=14.712653, z=69.248747, rx=0.007626, ry=-85.994743, rz=0.007244, shoulder=lefty, elbow=epositive, wrist=wpositive, fatherId=frmaster[1]}
  [295] = {x=99.242552, y=15.054876, z=66.008267, rx=-0.001359, ry=-84.105973, rz=-0.001065, shoulder=lefty, elbow=epositive, wrist=wpositive, fatherId=frmaster[1]}
  [296] = {x=101.001027, y=15.39368, z=62.930477, rx=-0.002933, ry=-82.347969, rz=-0.003321, shoulder=lefty, elbow=epositive, wrist=wpositive, fatherId=frmaster[1]}
  [297] = {x=102.722247, y=15.712182, z=59.655074, rx=-0.001305, ry=-80.506151, rz=-0.001552, shoulder=lefty, elbow=epositive, wrist=wpositive, fatherId=frmaster[1]}
  [298] = {x=104.194124, y=16.026632, z=56.594297, rx=0.005433, ry=-78.81259, rz=0.004583, shoulder=lefty, elbow=epositive, wrist=wpositive, fatherId=frmaster[1]}
  [299] = {x=104.267493, y=17.20804, z=54.349504, rx=-0.00147, ry=-77.582363, rz=-0.001735, shoulder=lefty, elbow=epositive, wrist=wpositive, fatherId=frmaster[1]}
  [300] = {x=103.069943, y=18.308821, z=54.347974, rx=0.000976, ry=-77.582651, rz=0.000694, shoulder=lefty, elbow=epositive, wrist=wpositive, fatherId=frmaster[1]}
  [301] = {x=101.813283, y=19.354473, z=54.355792, rx=-0.001279, ry=-77.581608, rz=-0.001159, shoulder=lefty, elbow=epositive, wrist=wpositive, fatherId=frmaster[1]}
  [302] = {x=100.510733, y=20.329976, z=54.350841, rx=0.002819, ry=-77.581863, rz=0.002541, shoulder=lefty, elbow=epositive, wrist=wpositive, fatherId=frmaster[1]}
  [303] = {x=99.207651, y=21.310883, z=54.348007, rx=0.002932, ry=-77.582776, rz=0.002519, shoulder=lefty, elbow=epositive, wrist=wpositive, fatherId=frmaster[1]}
  [304] = {x=97.868036, y=22.255333, z=54.355511, rx=-0.000825, ry=-77.581281, rz=-0.0007, shoulder=lefty, elbow=epositive, wrist=wpositive, fatherId=frmaster[1]}
  [305] = {x=96.529068, y=23.197406, z=54.35321, rx=-0.002023, ry=-77.582158, rz=-0.00165, shoulder=lefty, elbow=epositive, wrist=wpositive, fatherId=frmaster[1]}
